   // UNICODE_TO_GBK[37326] := 16#941A;
   // UNICODE_TO_GBK[37327] := 16#E78C;
   // UNICODE_TO_GBK[37328] := 16#941B;
   // UNICODE_TO_GBK[37329] := 16#E78D;
   // UNICODE_TO_GBK[37330] := 16#941C;
   // UNICODE_TO_GBK[37331] := 16#E78E;
   // UNICODE_TO_GBK[37332] := 16#941D;
   // UNICODE_TO_GBK[37333] := 16#E78F;
   // UNICODE_TO_GBK[37334] := 16#941E;
   // UNICODE_TO_GBK[37335] := 16#E790;
   // UNICODE_TO_GBK[37336] := 16#941F;
   // UNICODE_TO_GBK[37337] := 16#E791;
   // UNICODE_TO_GBK[37338] := 16#9420;
   // UNICODE_TO_GBK[37339] := 16#E792;
   // UNICODE_TO_GBK[37340] := 16#9421;
   // UNICODE_TO_GBK[37341] := 16#E793;
   // UNICODE_TO_GBK[37342] := 16#9422;
   // UNICODE_TO_GBK[37343] := 16#E794;
   // UNICODE_TO_GBK[37344] := 16#9423;
   // UNICODE_TO_GBK[37345] := 16#E795;
   // UNICODE_TO_GBK[37346] := 16#9424;
   // UNICODE_TO_GBK[37347] := 16#E796;
   // UNICODE_TO_GBK[37348] := 16#9425;
   // UNICODE_TO_GBK[37349] := 16#E797;
   // UNICODE_TO_GBK[37350] := 16#9426;
   // UNICODE_TO_GBK[37351] := 16#E798;
   // UNICODE_TO_GBK[37352] := 16#9427;
   // UNICODE_TO_GBK[37353] := 16#E799;
   // UNICODE_TO_GBK[37354] := 16#9428;
   // UNICODE_TO_GBK[37355] := 16#E79A;
   // UNICODE_TO_GBK[37356] := 16#9429;
   // UNICODE_TO_GBK[37357] := 16#E79B;
   // UNICODE_TO_GBK[37358] := 16#942A;
   // UNICODE_TO_GBK[37359] := 16#E79C;
   // UNICODE_TO_GBK[37360] := 16#942B;
   // UNICODE_TO_GBK[37361] := 16#E79D;
   // UNICODE_TO_GBK[37362] := 16#942C;
   // UNICODE_TO_GBK[37363] := 16#E79E;
   // UNICODE_TO_GBK[37364] := 16#942D;
   // UNICODE_TO_GBK[37365] := 16#E79F;
   // UNICODE_TO_GBK[37366] := 16#942E;
   // UNICODE_TO_GBK[37367] := 16#E7A0;
   // UNICODE_TO_GBK[37368] := 16#942F;
   // UNICODE_TO_GBK[37369] := 16#E840;
   // UNICODE_TO_GBK[37370] := 16#9430;
   // UNICODE_TO_GBK[37371] := 16#E841;
   // UNICODE_TO_GBK[37372] := 16#9431;
   // UNICODE_TO_GBK[37373] := 16#E842;
   // UNICODE_TO_GBK[37374] := 16#9432;
   // UNICODE_TO_GBK[37375] := 16#E843;
   // UNICODE_TO_GBK[37376] := 16#9433;
   // UNICODE_TO_GBK[37377] := 16#E844;
   // UNICODE_TO_GBK[37378] := 16#9434;
   // UNICODE_TO_GBK[37379] := 16#E845;
   // UNICODE_TO_GBK[37380] := 16#9435;
   // UNICODE_TO_GBK[37381] := 16#E846;
   // UNICODE_TO_GBK[37382] := 16#9436;
   // UNICODE_TO_GBK[37383] := 16#E847;
   // UNICODE_TO_GBK[37384] := 16#9437;
   // UNICODE_TO_GBK[37385] := 16#E848;
   // UNICODE_TO_GBK[37386] := 16#9438;
   // UNICODE_TO_GBK[37387] := 16#E849;
   // UNICODE_TO_GBK[37388] := 16#9439;
   // UNICODE_TO_GBK[37389] := 16#E84A;
   // UNICODE_TO_GBK[37390] := 16#943A;
   // UNICODE_TO_GBK[37391] := 16#E84B;
   // UNICODE_TO_GBK[37392] := 16#943B;
   // UNICODE_TO_GBK[37393] := 16#E84C;
   // UNICODE_TO_GBK[37394] := 16#943C;
   // UNICODE_TO_GBK[37395] := 16#E84D;
   // UNICODE_TO_GBK[37396] := 16#943D;
   // UNICODE_TO_GBK[37397] := 16#E84E;
   // UNICODE_TO_GBK[37398] := 16#943E;
   // UNICODE_TO_GBK[37399] := 16#F6CD;
   // UNICODE_TO_GBK[37400] := 16#943F;
   // UNICODE_TO_GBK[37401] := 16#E84F;
   // UNICODE_TO_GBK[37402] := 16#9440;
   // UNICODE_TO_GBK[37403] := 16#E850;
   // UNICODE_TO_GBK[37404] := 16#9441;
   // UNICODE_TO_GBK[37405] := 16#E851;
   // UNICODE_TO_GBK[37406] := 16#9442;
   // UNICODE_TO_GBK[37407] := 16#E852;
   // UNICODE_TO_GBK[37408] := 16#9443;
   // UNICODE_TO_GBK[37409] := 16#E853;
   // UNICODE_TO_GBK[37410] := 16#9444;
   // UNICODE_TO_GBK[37411] := 16#E854;
   // UNICODE_TO_GBK[37412] := 16#9445;
   // UNICODE_TO_GBK[37413] := 16#E855;
   // UNICODE_TO_GBK[37414] := 16#9446;
   // UNICODE_TO_GBK[37415] := 16#E856;
   // UNICODE_TO_GBK[37416] := 16#9447;
   // UNICODE_TO_GBK[37417] := 16#E857;
   // UNICODE_TO_GBK[37418] := 16#9448;
   // UNICODE_TO_GBK[37419] := 16#E858;
   // UNICODE_TO_GBK[37420] := 16#9449;
   // UNICODE_TO_GBK[37421] := 16#E859;
   // UNICODE_TO_GBK[37422] := 16#944A;
   // UNICODE_TO_GBK[37423] := 16#E85A;
   // UNICODE_TO_GBK[37424] := 16#944B;
   // UNICODE_TO_GBK[37425] := 16#E85B;
   // UNICODE_TO_GBK[37426] := 16#944C;
   // UNICODE_TO_GBK[37427] := 16#E85C;
   // UNICODE_TO_GBK[37428] := 16#944D;
   // UNICODE_TO_GBK[37429] := 16#E85D;
   // UNICODE_TO_GBK[37430] := 16#944E;
   // UNICODE_TO_GBK[37431] := 16#E85E;
   // UNICODE_TO_GBK[37432] := 16#944F;
   // UNICODE_TO_GBK[37433] := 16#E85F;
   // UNICODE_TO_GBK[37434] := 16#9450;
   // UNICODE_TO_GBK[37435] := 16#E860;
   // UNICODE_TO_GBK[37436] := 16#9451;
   // UNICODE_TO_GBK[37437] := 16#E861;
   // UNICODE_TO_GBK[37438] := 16#9452;
   // UNICODE_TO_GBK[37439] := 16#E862;
   // UNICODE_TO_GBK[37440] := 16#9453;
   // UNICODE_TO_GBK[37441] := 16#E863;
   // UNICODE_TO_GBK[37442] := 16#9454;
   // UNICODE_TO_GBK[37443] := 16#E864;
   // UNICODE_TO_GBK[37444] := 16#9455;
   // UNICODE_TO_GBK[37445] := 16#E865;
   // UNICODE_TO_GBK[37446] := 16#9456;
   // UNICODE_TO_GBK[37447] := 16#E866;
   // UNICODE_TO_GBK[37448] := 16#9457;
   // UNICODE_TO_GBK[37449] := 16#E867;
   // UNICODE_TO_GBK[37450] := 16#9458;
   // UNICODE_TO_GBK[37451] := 16#E868;
   // UNICODE_TO_GBK[37452] := 16#9459;
   // UNICODE_TO_GBK[37453] := 16#E869;
   // UNICODE_TO_GBK[37454] := 16#945A;
   // UNICODE_TO_GBK[37455] := 16#E86A;
   // UNICODE_TO_GBK[37456] := 16#945B;
   // UNICODE_TO_GBK[37457] := 16#E86B;
   // UNICODE_TO_GBK[37458] := 16#945C;
   // UNICODE_TO_GBK[37459] := 16#E86C;
   // UNICODE_TO_GBK[37460] := 16#945D;
   // UNICODE_TO_GBK[37461] := 16#E86D;
   // UNICODE_TO_GBK[37462] := 16#945E;
   // UNICODE_TO_GBK[37463] := 16#E86E;
   // UNICODE_TO_GBK[37464] := 16#945F;
   // UNICODE_TO_GBK[37465] := 16#E86F;
   // UNICODE_TO_GBK[37466] := 16#9460;
   // UNICODE_TO_GBK[37467] := 16#E870;
   // UNICODE_TO_GBK[37468] := 16#9461;
   // UNICODE_TO_GBK[37469] := 16#E871;
   // UNICODE_TO_GBK[37470] := 16#9462;
   // UNICODE_TO_GBK[37471] := 16#E872;
   // UNICODE_TO_GBK[37472] := 16#9463;
   // UNICODE_TO_GBK[37473] := 16#E873;
   // UNICODE_TO_GBK[37474] := 16#9464;
   // UNICODE_TO_GBK[37475] := 16#E874;
   // UNICODE_TO_GBK[37476] := 16#9465;
   // UNICODE_TO_GBK[37477] := 16#E875;
   // UNICODE_TO_GBK[37478] := 16#9466;
   // UNICODE_TO_GBK[37479] := 16#E876;
   // UNICODE_TO_GBK[37480] := 16#9467;
   // UNICODE_TO_GBK[37481] := 16#E877;
   // UNICODE_TO_GBK[37482] := 16#9468;
   // UNICODE_TO_GBK[37483] := 16#E878;
   // UNICODE_TO_GBK[37484] := 16#9469;
   // UNICODE_TO_GBK[37485] := 16#E879;
   // UNICODE_TO_GBK[37486] := 16#946A;
   // UNICODE_TO_GBK[37487] := 16#E87A;
   // UNICODE_TO_GBK[37488] := 16#946B;
   // UNICODE_TO_GBK[37489] := 16#F6CE;
   // UNICODE_TO_GBK[37490] := 16#946C;
   // UNICODE_TO_GBK[37491] := 16#E87B;
   // UNICODE_TO_GBK[37492] := 16#946D;
   // UNICODE_TO_GBK[37493] := 16#E87C;
   // UNICODE_TO_GBK[37494] := 16#946E;
   // UNICODE_TO_GBK[37495] := 16#E87D;
   // UNICODE_TO_GBK[37496] := 16#946F;
   // UNICODE_TO_GBK[37497] := 16#E87E;
   // UNICODE_TO_GBK[37498] := 16#9470;
   // UNICODE_TO_GBK[37499] := 16#E880;
   // UNICODE_TO_GBK[37500] := 16#9471;
   // UNICODE_TO_GBK[37501] := 16#E881;
   // UNICODE_TO_GBK[37502] := 16#9472;
   // UNICODE_TO_GBK[37503] := 16#E882;
   // UNICODE_TO_GBK[37504] := 16#9473;
   // UNICODE_TO_GBK[37505] := 16#E883;
   // UNICODE_TO_GBK[37506] := 16#9474;
   // UNICODE_TO_GBK[37507] := 16#E884;
   // UNICODE_TO_GBK[37508] := 16#9475;
   // UNICODE_TO_GBK[37509] := 16#E885;
   // UNICODE_TO_GBK[37510] := 16#9476;
   // UNICODE_TO_GBK[37511] := 16#E886;
   // UNICODE_TO_GBK[37512] := 16#9477;
   // UNICODE_TO_GBK[37513] := 16#E887;
   // UNICODE_TO_GBK[37514] := 16#9478;
   // UNICODE_TO_GBK[37515] := 16#E888;
   // UNICODE_TO_GBK[37516] := 16#9479;
   // UNICODE_TO_GBK[37517] := 16#E889;
   // UNICODE_TO_GBK[37518] := 16#947A;
   // UNICODE_TO_GBK[37519] := 16#E88A;
   // UNICODE_TO_GBK[37520] := 16#947B;
   // UNICODE_TO_GBK[37521] := 16#E88B;
   // UNICODE_TO_GBK[37522] := 16#947C;
   // UNICODE_TO_GBK[37523] := 16#E88C;
   // UNICODE_TO_GBK[37524] := 16#947D;
   // UNICODE_TO_GBK[37525] := 16#E88D;
   // UNICODE_TO_GBK[37526] := 16#947E;
   // UNICODE_TO_GBK[37527] := 16#E88E;
   // UNICODE_TO_GBK[37528] := 16#947F;
   // UNICODE_TO_GBK[37529] := 16#E88F;
   // UNICODE_TO_GBK[37530] := 16#9480;
   // UNICODE_TO_GBK[37531] := 16#E890;
   // UNICODE_TO_GBK[37532] := 16#9481;
   // UNICODE_TO_GBK[37533] := 16#E891;
   // UNICODE_TO_GBK[37534] := 16#9482;
   // UNICODE_TO_GBK[37535] := 16#E892;
   // UNICODE_TO_GBK[37536] := 16#9483;
   // UNICODE_TO_GBK[37537] := 16#E893;
   // UNICODE_TO_GBK[37538] := 16#9484;
   // UNICODE_TO_GBK[37539] := 16#E894;
   // UNICODE_TO_GBK[37540] := 16#9485;
   // UNICODE_TO_GBK[37541] := 16#EEC4;
   // UNICODE_TO_GBK[37542] := 16#9486;
   // UNICODE_TO_GBK[37543] := 16#EEC5;
   // UNICODE_TO_GBK[37544] := 16#9487;
   // UNICODE_TO_GBK[37545] := 16#EEC6;
   // UNICODE_TO_GBK[37546] := 16#9488;
   // UNICODE_TO_GBK[37547] := 16#D5EB;
   // UNICODE_TO_GBK[37548] := 16#9489;
   // UNICODE_TO_GBK[37549] := 16#B6A4;
   // UNICODE_TO_GBK[37550] := 16#948A;
   // UNICODE_TO_GBK[37551] := 16#EEC8;
   // UNICODE_TO_GBK[37552] := 16#948B;
   // UNICODE_TO_GBK[37553] := 16#EEC7;
   // UNICODE_TO_GBK[37554] := 16#948C;
   // UNICODE_TO_GBK[37555] := 16#EEC9;
   // UNICODE_TO_GBK[37556] := 16#948D;
   // UNICODE_TO_GBK[37557] := 16#EECA;
   // UNICODE_TO_GBK[37558] := 16#948E;
   // UNICODE_TO_GBK[37559] := 16#C7A5;
   // UNICODE_TO_GBK[37560] := 16#948F;
   // UNICODE_TO_GBK[37561] := 16#EECB;
   // UNICODE_TO_GBK[37562] := 16#9490;
   // UNICODE_TO_GBK[37563] := 16#EECC;
   // UNICODE_TO_GBK[37564] := 16#9491;
   // UNICODE_TO_GBK[37565] := 16#E895;
   // UNICODE_TO_GBK[37566] := 16#9492;
   // UNICODE_TO_GBK[37567] := 16#B7B0;
   // UNICODE_TO_GBK[37568] := 16#9493;
   // UNICODE_TO_GBK[37569] := 16#B5F6;
   // UNICODE_TO_GBK[37570] := 16#9494;
   // UNICODE_TO_GBK[37571] := 16#EECD;
   // UNICODE_TO_GBK[37572] := 16#9495;
   // UNICODE_TO_GBK[37573] := 16#EECF;
   // UNICODE_TO_GBK[37574] := 16#9496;
   // UNICODE_TO_GBK[37575] := 16#E896;
   // UNICODE_TO_GBK[37576] := 16#9497;
   // UNICODE_TO_GBK[37577] := 16#EECE;
   // UNICODE_TO_GBK[37578] := 16#9498;
   // UNICODE_TO_GBK[37579] := 16#E897;
   // UNICODE_TO_GBK[37580] := 16#9499;
   // UNICODE_TO_GBK[37581] := 16#B8C6;
   // UNICODE_TO_GBK[37582] := 16#949A;
   // UNICODE_TO_GBK[37583] := 16#EED0;
   // UNICODE_TO_GBK[37584] := 16#949B;
   // UNICODE_TO_GBK[37585] := 16#EED1;
   // UNICODE_TO_GBK[37586] := 16#949C;
   // UNICODE_TO_GBK[37587] := 16#EED2;
   // UNICODE_TO_GBK[37588] := 16#949D;
   // UNICODE_TO_GBK[37589] := 16#B6DB;
   // UNICODE_TO_GBK[37590] := 16#949E;
   // UNICODE_TO_GBK[37591] := 16#B3AE;
   // UNICODE_TO_GBK[37592] := 16#949F;
   // UNICODE_TO_GBK[37593] := 16#D6D3;
   // UNICODE_TO_GBK[37594] := 16#94A0;
   // UNICODE_TO_GBK[37595] := 16#C4C6;
   // UNICODE_TO_GBK[37596] := 16#94A1;
   // UNICODE_TO_GBK[37597] := 16#B1B5;
   // UNICODE_TO_GBK[37598] := 16#94A2;
   // UNICODE_TO_GBK[37599] := 16#B8D6;
   // UNICODE_TO_GBK[37600] := 16#94A3;
   // UNICODE_TO_GBK[37601] := 16#EED3;
   // UNICODE_TO_GBK[37602] := 16#94A4;
   // UNICODE_TO_GBK[37603] := 16#EED4;
   // UNICODE_TO_GBK[37604] := 16#94A5;
   // UNICODE_TO_GBK[37605] := 16#D4BF;
   // UNICODE_TO_GBK[37606] := 16#94A6;
   // UNICODE_TO_GBK[37607] := 16#C7D5;
   // UNICODE_TO_GBK[37608] := 16#94A7;
   // UNICODE_TO_GBK[37609] := 16#BEFB;
   // UNICODE_TO_GBK[37610] := 16#94A8;
   // UNICODE_TO_GBK[37611] := 16#CED9;
   // UNICODE_TO_GBK[37612] := 16#94A9;
   // UNICODE_TO_GBK[37613] := 16#B9B3;
   // UNICODE_TO_GBK[37614] := 16#94AA;
   // UNICODE_TO_GBK[37615] := 16#EED6;
   // UNICODE_TO_GBK[37616] := 16#94AB;
   // UNICODE_TO_GBK[37617] := 16#EED5;
   // UNICODE_TO_GBK[37618] := 16#94AC;
   // UNICODE_TO_GBK[37619] := 16#EED8;
   // UNICODE_TO_GBK[37620] := 16#94AD;
   // UNICODE_TO_GBK[37621] := 16#EED7;
   // UNICODE_TO_GBK[37622] := 16#94AE;
   // UNICODE_TO_GBK[37623] := 16#C5A5;
   // UNICODE_TO_GBK[37624] := 16#94AF;
   // UNICODE_TO_GBK[37625] := 16#EED9;
   // UNICODE_TO_GBK[37626] := 16#94B0;
   // UNICODE_TO_GBK[37627] := 16#EEDA;
   // UNICODE_TO_GBK[37628] := 16#94B1;
   // UNICODE_TO_GBK[37629] := 16#C7AE;
   // UNICODE_TO_GBK[37630] := 16#94B2;
   // UNICODE_TO_GBK[37631] := 16#EEDB;
   // UNICODE_TO_GBK[37632] := 16#94B3;
   // UNICODE_TO_GBK[37633] := 16#C7AF;
   // UNICODE_TO_GBK[37634] := 16#94B4;
   // UNICODE_TO_GBK[37635] := 16#EEDC;
   // UNICODE_TO_GBK[37636] := 16#94B5;
   // UNICODE_TO_GBK[37637] := 16#B2A7;
   // UNICODE_TO_GBK[37638] := 16#94B6;
   // UNICODE_TO_GBK[37639] := 16#EEDD;
   // UNICODE_TO_GBK[37640] := 16#94B7;
   // UNICODE_TO_GBK[37641] := 16#EEDE;
   // UNICODE_TO_GBK[37642] := 16#94B8;
   // UNICODE_TO_GBK[37643] := 16#EEDF;
   // UNICODE_TO_GBK[37644] := 16#94B9;
   // UNICODE_TO_GBK[37645] := 16#EEE0;
   // UNICODE_TO_GBK[37646] := 16#94BA;
   // UNICODE_TO_GBK[37647] := 16#EEE1;
   // UNICODE_TO_GBK[37648] := 16#94BB;
   // UNICODE_TO_GBK[37649] := 16#D7EA;
   // UNICODE_TO_GBK[37650] := 16#94BC;
   // UNICODE_TO_GBK[37651] := 16#EEE2;
   // UNICODE_TO_GBK[37652] := 16#94BD;
   // UNICODE_TO_GBK[37653] := 16#EEE3;
   // UNICODE_TO_GBK[37654] := 16#94BE;
   // UNICODE_TO_GBK[37655] := 16#BCD8;
   // UNICODE_TO_GBK[37656] := 16#94BF;
   // UNICODE_TO_GBK[37657] := 16#EEE4;
   // UNICODE_TO_GBK[37658] := 16#94C0;
   // UNICODE_TO_GBK[37659] := 16#D3CB;
   // UNICODE_TO_GBK[37660] := 16#94C1;
   // UNICODE_TO_GBK[37661] := 16#CCFA;
   // UNICODE_TO_GBK[37662] := 16#94C2;
   // UNICODE_TO_GBK[37663] := 16#B2AC;
   // UNICODE_TO_GBK[37664] := 16#94C3;
   // UNICODE_TO_GBK[37665] := 16#C1E5;
   // UNICODE_TO_GBK[37666] := 16#94C4;
   // UNICODE_TO_GBK[37667] := 16#EEE5;
   // UNICODE_TO_GBK[37668] := 16#94C5;
   // UNICODE_TO_GBK[37669] := 16#C7A6;
   // UNICODE_TO_GBK[37670] := 16#94C6;
   // UNICODE_TO_GBK[37671] := 16#C3AD;
   // UNICODE_TO_GBK[37672] := 16#94C7;
   // UNICODE_TO_GBK[37673] := 16#E898;
   // UNICODE_TO_GBK[37674] := 16#94C8;
   // UNICODE_TO_GBK[37675] := 16#EEE6;
   // UNICODE_TO_GBK[37676] := 16#94C9;
   // UNICODE_TO_GBK[37677] := 16#EEE7;
   // UNICODE_TO_GBK[37678] := 16#94CA;
   // UNICODE_TO_GBK[37679] := 16#EEE8;
   // UNICODE_TO_GBK[37680] := 16#94CB;
   // UNICODE_TO_GBK[37681] := 16#EEE9;
   // UNICODE_TO_GBK[37682] := 16#94CC;
   // UNICODE_TO_GBK[37683] := 16#EEEA;
   // UNICODE_TO_GBK[37684] := 16#94CD;
   // UNICODE_TO_GBK[37685] := 16#EEEB;
   // UNICODE_TO_GBK[37686] := 16#94CE;
   // UNICODE_TO_GBK[37687] := 16#EEEC;
   // UNICODE_TO_GBK[37688] := 16#94CF;
   // UNICODE_TO_GBK[37689] := 16#E899;
   // UNICODE_TO_GBK[37690] := 16#94D0;
   // UNICODE_TO_GBK[37691] := 16#EEED;
   // UNICODE_TO_GBK[37692] := 16#94D1;
   // UNICODE_TO_GBK[37693] := 16#EEEE;
   // UNICODE_TO_GBK[37694] := 16#94D2;
   // UNICODE_TO_GBK[37695] := 16#EEEF;
   // UNICODE_TO_GBK[37696] := 16#94D3;
   // UNICODE_TO_GBK[37697] := 16#E89A;
   // UNICODE_TO_GBK[37698] := 16#94D4;
   // UNICODE_TO_GBK[37699] := 16#E89B;
   // UNICODE_TO_GBK[37700] := 16#94D5;
   // UNICODE_TO_GBK[37701] := 16#EEF0;
   // UNICODE_TO_GBK[37702] := 16#94D6;
   // UNICODE_TO_GBK[37703] := 16#EEF1;
   // UNICODE_TO_GBK[37704] := 16#94D7;
   // UNICODE_TO_GBK[37705] := 16#EEF2;
   // UNICODE_TO_GBK[37706] := 16#94D8;
   // UNICODE_TO_GBK[37707] := 16#EEF4;
   // UNICODE_TO_GBK[37708] := 16#94D9;
   // UNICODE_TO_GBK[37709] := 16#EEF3;
   // UNICODE_TO_GBK[37710] := 16#94DA;
   // UNICODE_TO_GBK[37711] := 16#E89C;
   // UNICODE_TO_GBK[37712] := 16#94DB;
   // UNICODE_TO_GBK[37713] := 16#EEF5;
   // UNICODE_TO_GBK[37714] := 16#94DC;
   // UNICODE_TO_GBK[37715] := 16#CDAD;
   // UNICODE_TO_GBK[37716] := 16#94DD;
   // UNICODE_TO_GBK[37717] := 16#C2C1;
   // UNICODE_TO_GBK[37718] := 16#94DE;
   // UNICODE_TO_GBK[37719] := 16#EEF6;
   // UNICODE_TO_GBK[37720] := 16#94DF;
   // UNICODE_TO_GBK[37721] := 16#EEF7;
   // UNICODE_TO_GBK[37722] := 16#94E0;
   // UNICODE_TO_GBK[37723] := 16#EEF8;
   // UNICODE_TO_GBK[37724] := 16#94E1;
   // UNICODE_TO_GBK[37725] := 16#D5A1;
   // UNICODE_TO_GBK[37726] := 16#94E2;
   // UNICODE_TO_GBK[37727] := 16#EEF9;
   // UNICODE_TO_GBK[37728] := 16#94E3;
   // UNICODE_TO_GBK[37729] := 16#CFB3;
   // UNICODE_TO_GBK[37730] := 16#94E4;
   // UNICODE_TO_GBK[37731] := 16#EEFA;
   // UNICODE_TO_GBK[37732] := 16#94E5;
   // UNICODE_TO_GBK[37733] := 16#EEFB;
   // UNICODE_TO_GBK[37734] := 16#94E6;
   // UNICODE_TO_GBK[37735] := 16#E89D;
   // UNICODE_TO_GBK[37736] := 16#94E7;
   // UNICODE_TO_GBK[37737] := 16#EEFC;
   // UNICODE_TO_GBK[37738] := 16#94E8;
   // UNICODE_TO_GBK[37739] := 16#EEFD;
   // UNICODE_TO_GBK[37740] := 16#94E9;
   // UNICODE_TO_GBK[37741] := 16#EFA1;
   // UNICODE_TO_GBK[37742] := 16#94EA;
   // UNICODE_TO_GBK[37743] := 16#EEFE;
   // UNICODE_TO_GBK[37744] := 16#94EB;
   // UNICODE_TO_GBK[37745] := 16#EFA2;
   // UNICODE_TO_GBK[37746] := 16#94EC;
   // UNICODE_TO_GBK[37747] := 16#B8F5;
   // UNICODE_TO_GBK[37748] := 16#94ED;
   // UNICODE_TO_GBK[37749] := 16#C3FA;
   // UNICODE_TO_GBK[37750] := 16#94EE;
   // UNICODE_TO_GBK[37751] := 16#EFA3;
   // UNICODE_TO_GBK[37752] := 16#94EF;
   // UNICODE_TO_GBK[37753] := 16#EFA4;
   // UNICODE_TO_GBK[37754] := 16#94F0;
   // UNICODE_TO_GBK[37755] := 16#BDC2;
   // UNICODE_TO_GBK[37756] := 16#94F1;
   // UNICODE_TO_GBK[37757] := 16#D2BF;
   // UNICODE_TO_GBK[37758] := 16#94F2;
   // UNICODE_TO_GBK[37759] := 16#B2F9;
   // UNICODE_TO_GBK[37760] := 16#94F3;
   // UNICODE_TO_GBK[37761] := 16#EFA5;
   // UNICODE_TO_GBK[37762] := 16#94F4;
   // UNICODE_TO_GBK[37763] := 16#EFA6;
   // UNICODE_TO_GBK[37764] := 16#94F5;
   // UNICODE_TO_GBK[37765] := 16#EFA7;
   // UNICODE_TO_GBK[37766] := 16#94F6;
   // UNICODE_TO_GBK[37767] := 16#D2F8;
   // UNICODE_TO_GBK[37768] := 16#94F7;
   // UNICODE_TO_GBK[37769] := 16#EFA8;
   // UNICODE_TO_GBK[37770] := 16#94F8;
   // UNICODE_TO_GBK[37771] := 16#D6FD;
   // UNICODE_TO_GBK[37772] := 16#94F9;
   // UNICODE_TO_GBK[37773] := 16#EFA9;
   // UNICODE_TO_GBK[37774] := 16#94FA;
   // UNICODE_TO_GBK[37775] := 16#C6CC;
   // UNICODE_TO_GBK[37776] := 16#94FB;
   // UNICODE_TO_GBK[37777] := 16#E89E;
   // UNICODE_TO_GBK[37778] := 16#94FC;
   // UNICODE_TO_GBK[37779] := 16#EFAA;
   // UNICODE_TO_GBK[37780] := 16#94FD;
   // UNICODE_TO_GBK[37781] := 16#EFAB;
   // UNICODE_TO_GBK[37782] := 16#94FE;
   // UNICODE_TO_GBK[37783] := 16#C1B4;
   // UNICODE_TO_GBK[37784] := 16#94FF;
   // UNICODE_TO_GBK[37785] := 16#EFAC;
   // UNICODE_TO_GBK[37786] := 16#9500;
   // UNICODE_TO_GBK[37787] := 16#CFFA;
   // UNICODE_TO_GBK[37788] := 16#9501;
   // UNICODE_TO_GBK[37789] := 16#CBF8;
   // UNICODE_TO_GBK[37790] := 16#9502;
   // UNICODE_TO_GBK[37791] := 16#EFAE;
   // UNICODE_TO_GBK[37792] := 16#9503;
   // UNICODE_TO_GBK[37793] := 16#EFAD;
   // UNICODE_TO_GBK[37794] := 16#9504;
   // UNICODE_TO_GBK[37795] := 16#B3FA;
   // UNICODE_TO_GBK[37796] := 16#9505;
   // UNICODE_TO_GBK[37797] := 16#B9F8;
   // UNICODE_TO_GBK[37798] := 16#9506;
   // UNICODE_TO_GBK[37799] := 16#EFAF;
   // UNICODE_TO_GBK[37800] := 16#9507;
   // UNICODE_TO_GBK[37801] := 16#EFB0;
   // UNICODE_TO_GBK[37802] := 16#9508;
   // UNICODE_TO_GBK[37803] := 16#D0E2;
   // UNICODE_TO_GBK[37804] := 16#9509;
   // UNICODE_TO_GBK[37805] := 16#EFB1;
   // UNICODE_TO_GBK[37806] := 16#950A;
   // UNICODE_TO_GBK[37807] := 16#EFB2;
   // UNICODE_TO_GBK[37808] := 16#950B;
   // UNICODE_TO_GBK[37809] := 16#B7E6;
   // UNICODE_TO_GBK[37810] := 16#950C;
   // UNICODE_TO_GBK[37811] := 16#D0BF;
   // UNICODE_TO_GBK[37812] := 16#950D;
   // UNICODE_TO_GBK[37813] := 16#EFB3;
   // UNICODE_TO_GBK[37814] := 16#950E;
   // UNICODE_TO_GBK[37815] := 16#EFB4;
   // UNICODE_TO_GBK[37816] := 16#950F;
   // UNICODE_TO_GBK[37817] := 16#EFB5;
   // UNICODE_TO_GBK[37818] := 16#9510;
   // UNICODE_TO_GBK[37819] := 16#C8F1;
   // UNICODE_TO_GBK[37820] := 16#9511;
   // UNICODE_TO_GBK[37821] := 16#CCE0;
   // UNICODE_TO_GBK[37822] := 16#9512;
   // UNICODE_TO_GBK[37823] := 16#EFB6;
   // UNICODE_TO_GBK[37824] := 16#9513;
   // UNICODE_TO_GBK[37825] := 16#EFB7;
   // UNICODE_TO_GBK[37826] := 16#9514;
   // UNICODE_TO_GBK[37827] := 16#EFB8;
   // UNICODE_TO_GBK[37828] := 16#9515;
   // UNICODE_TO_GBK[37829] := 16#EFB9;
   // UNICODE_TO_GBK[37830] := 16#9516;
   // UNICODE_TO_GBK[37831] := 16#EFBA;
   // UNICODE_TO_GBK[37832] := 16#9517;
   // UNICODE_TO_GBK[37833] := 16#D5E0;
   // UNICODE_TO_GBK[37834] := 16#9518;
   // UNICODE_TO_GBK[37835] := 16#EFBB;
   // UNICODE_TO_GBK[37836] := 16#9519;
   // UNICODE_TO_GBK[37837] := 16#B4ED;
   // UNICODE_TO_GBK[37838] := 16#951A;
   // UNICODE_TO_GBK[37839] := 16#C3AA;
   // UNICODE_TO_GBK[37840] := 16#951B;
   // UNICODE_TO_GBK[37841] := 16#EFBC;
   // UNICODE_TO_GBK[37842] := 16#951C;
   // UNICODE_TO_GBK[37843] := 16#E89F;
   // UNICODE_TO_GBK[37844] := 16#951D;
   // UNICODE_TO_GBK[37845] := 16#EFBD;
   // UNICODE_TO_GBK[37846] := 16#951E;
   // UNICODE_TO_GBK[37847] := 16#EFBE;
   // UNICODE_TO_GBK[37848] := 16#951F;
   // UNICODE_TO_GBK[37849] := 16#EFBF;
   // UNICODE_TO_GBK[37850] := 16#9520;
   // UNICODE_TO_GBK[37851] := 16#E8A0;
   // UNICODE_TO_GBK[37852] := 16#9521;
   // UNICODE_TO_GBK[37853] := 16#CEFD;
   // UNICODE_TO_GBK[37854] := 16#9522;
   // UNICODE_TO_GBK[37855] := 16#EFC0;
   // UNICODE_TO_GBK[37856] := 16#9523;
   // UNICODE_TO_GBK[37857] := 16#C2E0;
   // UNICODE_TO_GBK[37858] := 16#9524;
   // UNICODE_TO_GBK[37859] := 16#B4B8;
   // UNICODE_TO_GBK[37860] := 16#9525;
   // UNICODE_TO_GBK[37861] := 16#D7B6;
   // UNICODE_TO_GBK[37862] := 16#9526;
   // UNICODE_TO_GBK[37863] := 16#BDF5;
   // UNICODE_TO_GBK[37864] := 16#9527;
   // UNICODE_TO_GBK[37865] := 16#E940;
   // UNICODE_TO_GBK[37866] := 16#9528;
   // UNICODE_TO_GBK[37867] := 16#CFC7;
   // UNICODE_TO_GBK[37868] := 16#9529;
   // UNICODE_TO_GBK[37869] := 16#EFC3;
   // UNICODE_TO_GBK[37870] := 16#952A;
   // UNICODE_TO_GBK[37871] := 16#EFC1;
   // UNICODE_TO_GBK[37872] := 16#952B;
   // UNICODE_TO_GBK[37873] := 16#EFC2;
   // UNICODE_TO_GBK[37874] := 16#952C;
   // UNICODE_TO_GBK[37875] := 16#EFC4;
   // UNICODE_TO_GBK[37876] := 16#952D;
   // UNICODE_TO_GBK[37877] := 16#B6A7;
   // UNICODE_TO_GBK[37878] := 16#952E;
   // UNICODE_TO_GBK[37879] := 16#BCFC;
   // UNICODE_TO_GBK[37880] := 16#952F;
   // UNICODE_TO_GBK[37881] := 16#BEE2;
   // UNICODE_TO_GBK[37882] := 16#9530;
   // UNICODE_TO_GBK[37883] := 16#C3CC;
   // UNICODE_TO_GBK[37884] := 16#9531;
   // UNICODE_TO_GBK[37885] := 16#EFC5;
   // UNICODE_TO_GBK[37886] := 16#9532;
   // UNICODE_TO_GBK[37887] := 16#EFC6;
   // UNICODE_TO_GBK[37888] := 16#9533;
   // UNICODE_TO_GBK[37889] := 16#E941;
   // UNICODE_TO_GBK[37890] := 16#9534;
   // UNICODE_TO_GBK[37891] := 16#EFC7;
   // UNICODE_TO_GBK[37892] := 16#9535;
   // UNICODE_TO_GBK[37893] := 16#EFCF;
   // UNICODE_TO_GBK[37894] := 16#9536;
   // UNICODE_TO_GBK[37895] := 16#EFC8;
   // UNICODE_TO_GBK[37896] := 16#9537;
   // UNICODE_TO_GBK[37897] := 16#EFC9;
   // UNICODE_TO_GBK[37898] := 16#9538;
   // UNICODE_TO_GBK[37899] := 16#EFCA;
   // UNICODE_TO_GBK[37900] := 16#9539;
   // UNICODE_TO_GBK[37901] := 16#C7C2;
   // UNICODE_TO_GBK[37902] := 16#953A;
   // UNICODE_TO_GBK[37903] := 16#EFF1;
   // UNICODE_TO_GBK[37904] := 16#953B;
   // UNICODE_TO_GBK[37905] := 16#B6CD;
   // UNICODE_TO_GBK[37906] := 16#953C;
   // UNICODE_TO_GBK[37907] := 16#EFCB;
   // UNICODE_TO_GBK[37908] := 16#953D;
   // UNICODE_TO_GBK[37909] := 16#E942;
   // UNICODE_TO_GBK[37910] := 16#953E;
   // UNICODE_TO_GBK[37911] := 16#EFCC;
   // UNICODE_TO_GBK[37912] := 16#953F;
   // UNICODE_TO_GBK[37913] := 16#EFCD;
   // UNICODE_TO_GBK[37914] := 16#9540;
   // UNICODE_TO_GBK[37915] := 16#B6C6;
   // UNICODE_TO_GBK[37916] := 16#9541;
   // UNICODE_TO_GBK[37917] := 16#C3BE;
   // UNICODE_TO_GBK[37918] := 16#9542;
   // UNICODE_TO_GBK[37919] := 16#EFCE;
   // UNICODE_TO_GBK[37920] := 16#9543;
   // UNICODE_TO_GBK[37921] := 16#E943;
   // UNICODE_TO_GBK[37922] := 16#9544;
   // UNICODE_TO_GBK[37923] := 16#EFD0;
   // UNICODE_TO_GBK[37924] := 16#9545;
   // UNICODE_TO_GBK[37925] := 16#EFD1;
   // UNICODE_TO_GBK[37926] := 16#9546;
   // UNICODE_TO_GBK[37927] := 16#EFD2;
   // UNICODE_TO_GBK[37928] := 16#9547;
   // UNICODE_TO_GBK[37929] := 16#D5F2;
   // UNICODE_TO_GBK[37930] := 16#9548;
   // UNICODE_TO_GBK[37931] := 16#E944;
   // UNICODE_TO_GBK[37932] := 16#9549;
   // UNICODE_TO_GBK[37933] := 16#EFD3;
   // UNICODE_TO_GBK[37934] := 16#954A;
   // UNICODE_TO_GBK[37935] := 16#C4F7;
   // UNICODE_TO_GBK[37936] := 16#954B;
   // UNICODE_TO_GBK[37937] := 16#E945;
   // UNICODE_TO_GBK[37938] := 16#954C;
   // UNICODE_TO_GBK[37939] := 16#EFD4;
   // UNICODE_TO_GBK[37940] := 16#954D;
   // UNICODE_TO_GBK[37941] := 16#C4F8;
   // UNICODE_TO_GBK[37942] := 16#954E;
   // UNICODE_TO_GBK[37943] := 16#EFD5;
   // UNICODE_TO_GBK[37944] := 16#954F;
   // UNICODE_TO_GBK[37945] := 16#EFD6;
   // UNICODE_TO_GBK[37946] := 16#9550;
   // UNICODE_TO_GBK[37947] := 16#B8E4;
   // UNICODE_TO_GBK[37948] := 16#9551;
   // UNICODE_TO_GBK[37949] := 16#B0F7;
   // UNICODE_TO_GBK[37950] := 16#9552;
   // UNICODE_TO_GBK[37951] := 16#EFD7;
   // UNICODE_TO_GBK[37952] := 16#9553;
   // UNICODE_TO_GBK[37953] := 16#EFD8;
   // UNICODE_TO_GBK[37954] := 16#9554;
   // UNICODE_TO_GBK[37955] := 16#EFD9;
   // UNICODE_TO_GBK[37956] := 16#9555;
   // UNICODE_TO_GBK[37957] := 16#E946;
   // UNICODE_TO_GBK[37958] := 16#9556;
   // UNICODE_TO_GBK[37959] := 16#EFDA;
   // UNICODE_TO_GBK[37960] := 16#9557;
   // UNICODE_TO_GBK[37961] := 16#EFDB;
   // UNICODE_TO_GBK[37962] := 16#9558;
   // UNICODE_TO_GBK[37963] := 16#EFDC;
   // UNICODE_TO_GBK[37964] := 16#9559;
   // UNICODE_TO_GBK[37965] := 16#EFDD;
   // UNICODE_TO_GBK[37966] := 16#955A;
   // UNICODE_TO_GBK[37967] := 16#E947;
   // UNICODE_TO_GBK[37968] := 16#955B;
   // UNICODE_TO_GBK[37969] := 16#EFDE;
   // UNICODE_TO_GBK[37970] := 16#955C;
   // UNICODE_TO_GBK[37971] := 16#BEB5;
   // UNICODE_TO_GBK[37972] := 16#955D;
   // UNICODE_TO_GBK[37973] := 16#EFE1;
   // UNICODE_TO_GBK[37974] := 16#955E;
   // UNICODE_TO_GBK[37975] := 16#EFDF;
   // UNICODE_TO_GBK[37976] := 16#955F;
   // UNICODE_TO_GBK[37977] := 16#EFE0;
   // UNICODE_TO_GBK[37978] := 16#9560;
   // UNICODE_TO_GBK[37979] := 16#E948;
   // UNICODE_TO_GBK[37980] := 16#9561;
   // UNICODE_TO_GBK[37981] := 16#EFE2;
   // UNICODE_TO_GBK[37982] := 16#9562;
   // UNICODE_TO_GBK[37983] := 16#EFE3;
   // UNICODE_TO_GBK[37984] := 16#9563;
   // UNICODE_TO_GBK[37985] := 16#C1CD;
   // UNICODE_TO_GBK[37986] := 16#9564;
   // UNICODE_TO_GBK[37987] := 16#EFE4;
   // UNICODE_TO_GBK[37988] := 16#9565;
   // UNICODE_TO_GBK[37989] := 16#EFE5;
   // UNICODE_TO_GBK[37990] := 16#9566;
   // UNICODE_TO_GBK[37991] := 16#EFE6;
   // UNICODE_TO_GBK[37992] := 16#9567;
   // UNICODE_TO_GBK[37993] := 16#EFE7;
   // UNICODE_TO_GBK[37994] := 16#9568;
   // UNICODE_TO_GBK[37995] := 16#EFE8;
   // UNICODE_TO_GBK[37996] := 16#9569;
   // UNICODE_TO_GBK[37997] := 16#EFE9;
   // UNICODE_TO_GBK[37998] := 16#956A;
   // UNICODE_TO_GBK[37999] := 16#EFEA;
   // UNICODE_TO_GBK[38000] := 16#956B;
   // UNICODE_TO_GBK[38001] := 16#EFEB;
   // UNICODE_TO_GBK[38002] := 16#956C;
   // UNICODE_TO_GBK[38003] := 16#EFEC;
   // UNICODE_TO_GBK[38004] := 16#956D;
   // UNICODE_TO_GBK[38005] := 16#C0D8;
   // UNICODE_TO_GBK[38006] := 16#956E;
   // UNICODE_TO_GBK[38007] := 16#E949;
   // UNICODE_TO_GBK[38008] := 16#956F;
   // UNICODE_TO_GBK[38009] := 16#EFED;
   // UNICODE_TO_GBK[38010] := 16#9570;
   // UNICODE_TO_GBK[38011] := 16#C1AD;
   // UNICODE_TO_GBK[38012] := 16#9571;
   // UNICODE_TO_GBK[38013] := 16#EFEE;
   // UNICODE_TO_GBK[38014] := 16#9572;
   // UNICODE_TO_GBK[38015] := 16#EFEF;
   // UNICODE_TO_GBK[38016] := 16#9573;
   // UNICODE_TO_GBK[38017] := 16#EFF0;
   // UNICODE_TO_GBK[38018] := 16#9574;
   // UNICODE_TO_GBK[38019] := 16#E94A;
   // UNICODE_TO_GBK[38020] := 16#9575;
   // UNICODE_TO_GBK[38021] := 16#E94B;
   // UNICODE_TO_GBK[38022] := 16#9576;
   // UNICODE_TO_GBK[38023] := 16#CFE2;
   // UNICODE_TO_GBK[38024] := 16#9577;
   // UNICODE_TO_GBK[38025] := 16#E94C;
   // UNICODE_TO_GBK[38026] := 16#9578;
   // UNICODE_TO_GBK[38027] := 16#E94D;
   // UNICODE_TO_GBK[38028] := 16#9579;
   // UNICODE_TO_GBK[38029] := 16#E94E;
   // UNICODE_TO_GBK[38030] := 16#957A;
   // UNICODE_TO_GBK[38031] := 16#E94F;
   // UNICODE_TO_GBK[38032] := 16#957B;
   // UNICODE_TO_GBK[38033] := 16#E950;
   // UNICODE_TO_GBK[38034] := 16#957C;
   // UNICODE_TO_GBK[38035] := 16#E951;
   // UNICODE_TO_GBK[38036] := 16#957D;
   // UNICODE_TO_GBK[38037] := 16#E952;
   // UNICODE_TO_GBK[38038] := 16#957E;
   // UNICODE_TO_GBK[38039] := 16#E953;
   // UNICODE_TO_GBK[38040] := 16#957F;
   // UNICODE_TO_GBK[38041] := 16#B3A4;
   // UNICODE_TO_GBK[38042] := 16#9580;
   // UNICODE_TO_GBK[38043] := 16#E954;
   // UNICODE_TO_GBK[38044] := 16#9581;
   // UNICODE_TO_GBK[38045] := 16#E955;
   // UNICODE_TO_GBK[38046] := 16#9582;
   // UNICODE_TO_GBK[38047] := 16#E956;
   // UNICODE_TO_GBK[38048] := 16#9583;
   // UNICODE_TO_GBK[38049] := 16#E957;
   // UNICODE_TO_GBK[38050] := 16#9584;
   // UNICODE_TO_GBK[38051] := 16#E958;
   // UNICODE_TO_GBK[38052] := 16#9585;
   // UNICODE_TO_GBK[38053] := 16#E959;
   // UNICODE_TO_GBK[38054] := 16#9586;
   // UNICODE_TO_GBK[38055] := 16#E95A;
   // UNICODE_TO_GBK[38056] := 16#9587;
   // UNICODE_TO_GBK[38057] := 16#E95B;
   // UNICODE_TO_GBK[38058] := 16#9588;
   // UNICODE_TO_GBK[38059] := 16#E95C;
   // UNICODE_TO_GBK[38060] := 16#9589;
   // UNICODE_TO_GBK[38061] := 16#E95D;
   // UNICODE_TO_GBK[38062] := 16#958A;
   // UNICODE_TO_GBK[38063] := 16#E95E;
   // UNICODE_TO_GBK[38064] := 16#958B;
   // UNICODE_TO_GBK[38065] := 16#E95F;
   // UNICODE_TO_GBK[38066] := 16#958C;
   // UNICODE_TO_GBK[38067] := 16#E960;
   // UNICODE_TO_GBK[38068] := 16#958D;
   // UNICODE_TO_GBK[38069] := 16#E961;
   // UNICODE_TO_GBK[38070] := 16#958E;
   // UNICODE_TO_GBK[38071] := 16#E962;
   // UNICODE_TO_GBK[38072] := 16#958F;
   // UNICODE_TO_GBK[38073] := 16#E963;
   // UNICODE_TO_GBK[38074] := 16#9590;
   // UNICODE_TO_GBK[38075] := 16#E964;
   // UNICODE_TO_GBK[38076] := 16#9591;
   // UNICODE_TO_GBK[38077] := 16#E965;
   // UNICODE_TO_GBK[38078] := 16#9592;
   // UNICODE_TO_GBK[38079] := 16#E966;
   // UNICODE_TO_GBK[38080] := 16#9593;
   // UNICODE_TO_GBK[38081] := 16#E967;
   // UNICODE_TO_GBK[38082] := 16#9594;
   // UNICODE_TO_GBK[38083] := 16#E968;
   // UNICODE_TO_GBK[38084] := 16#9595;
   // UNICODE_TO_GBK[38085] := 16#E969;
   // UNICODE_TO_GBK[38086] := 16#9596;
   // UNICODE_TO_GBK[38087] := 16#E96A;
   // UNICODE_TO_GBK[38088] := 16#9597;
   // UNICODE_TO_GBK[38089] := 16#E96B;
   // UNICODE_TO_GBK[38090] := 16#9598;
   // UNICODE_TO_GBK[38091] := 16#E96C;
   // UNICODE_TO_GBK[38092] := 16#9599;
   // UNICODE_TO_GBK[38093] := 16#E96D;
   // UNICODE_TO_GBK[38094] := 16#959A;
   // UNICODE_TO_GBK[38095] := 16#E96E;
   // UNICODE_TO_GBK[38096] := 16#959B;
   // UNICODE_TO_GBK[38097] := 16#E96F;
   // UNICODE_TO_GBK[38098] := 16#959C;
   // UNICODE_TO_GBK[38099] := 16#E970;
   // UNICODE_TO_GBK[38100] := 16#959D;
   // UNICODE_TO_GBK[38101] := 16#E971;
   // UNICODE_TO_GBK[38102] := 16#959E;
   // UNICODE_TO_GBK[38103] := 16#E972;
   // UNICODE_TO_GBK[38104] := 16#959F;
   // UNICODE_TO_GBK[38105] := 16#E973;
   // UNICODE_TO_GBK[38106] := 16#95A0;
   // UNICODE_TO_GBK[38107] := 16#E974;
   // UNICODE_TO_GBK[38108] := 16#95A1;
   // UNICODE_TO_GBK[38109] := 16#E975;
   // UNICODE_TO_GBK[38110] := 16#95A2;
   // UNICODE_TO_GBK[38111] := 16#E976;
   // UNICODE_TO_GBK[38112] := 16#95A3;
   // UNICODE_TO_GBK[38113] := 16#E977;
   // UNICODE_TO_GBK[38114] := 16#95A4;
   // UNICODE_TO_GBK[38115] := 16#E978;
   // UNICODE_TO_GBK[38116] := 16#95A5;
   // UNICODE_TO_GBK[38117] := 16#E979;
   // UNICODE_TO_GBK[38118] := 16#95A6;
   // UNICODE_TO_GBK[38119] := 16#E97A;
   // UNICODE_TO_GBK[38120] := 16#95A7;
   // UNICODE_TO_GBK[38121] := 16#E97B;
   // UNICODE_TO_GBK[38122] := 16#95A8;
   // UNICODE_TO_GBK[38123] := 16#E97C;
   // UNICODE_TO_GBK[38124] := 16#95A9;
   // UNICODE_TO_GBK[38125] := 16#E97D;
   // UNICODE_TO_GBK[38126] := 16#95AA;
   // UNICODE_TO_GBK[38127] := 16#E97E;
   // UNICODE_TO_GBK[38128] := 16#95AB;
   // UNICODE_TO_GBK[38129] := 16#E980;
   // UNICODE_TO_GBK[38130] := 16#95AC;
   // UNICODE_TO_GBK[38131] := 16#E981;
   // UNICODE_TO_GBK[38132] := 16#95AD;
   // UNICODE_TO_GBK[38133] := 16#E982;
   // UNICODE_TO_GBK[38134] := 16#95AE;
   // UNICODE_TO_GBK[38135] := 16#E983;
   // UNICODE_TO_GBK[38136] := 16#95AF;
   // UNICODE_TO_GBK[38137] := 16#E984;
   // UNICODE_TO_GBK[38138] := 16#95B0;
   // UNICODE_TO_GBK[38139] := 16#E985;
   // UNICODE_TO_GBK[38140] := 16#95B1;
   // UNICODE_TO_GBK[38141] := 16#E986;
   // UNICODE_TO_GBK[38142] := 16#95B2;
   // UNICODE_TO_GBK[38143] := 16#E987;
   // UNICODE_TO_GBK[38144] := 16#95B3;
   // UNICODE_TO_GBK[38145] := 16#E988;
   // UNICODE_TO_GBK[38146] := 16#95B4;
   // UNICODE_TO_GBK[38147] := 16#E989;
   // UNICODE_TO_GBK[38148] := 16#95B5;
   // UNICODE_TO_GBK[38149] := 16#E98A;
   // UNICODE_TO_GBK[38150] := 16#95B6;
   // UNICODE_TO_GBK[38151] := 16#E98B;
   // UNICODE_TO_GBK[38152] := 16#95B7;
   // UNICODE_TO_GBK[38153] := 16#E98C;
   // UNICODE_TO_GBK[38154] := 16#95B8;
   // UNICODE_TO_GBK[38155] := 16#E98D;
   // UNICODE_TO_GBK[38156] := 16#95B9;
   // UNICODE_TO_GBK[38157] := 16#E98E;
   // UNICODE_TO_GBK[38158] := 16#95BA;
   // UNICODE_TO_GBK[38159] := 16#E98F;
   // UNICODE_TO_GBK[38160] := 16#95BB;
   // UNICODE_TO_GBK[38161] := 16#E990;
   // UNICODE_TO_GBK[38162] := 16#95BC;
   // UNICODE_TO_GBK[38163] := 16#E991;
   // UNICODE_TO_GBK[38164] := 16#95BD;
   // UNICODE_TO_GBK[38165] := 16#E992;
   // UNICODE_TO_GBK[38166] := 16#95BE;
   // UNICODE_TO_GBK[38167] := 16#E993;
   // UNICODE_TO_GBK[38168] := 16#95BF;
   // UNICODE_TO_GBK[38169] := 16#E994;
   // UNICODE_TO_GBK[38170] := 16#95C0;
   // UNICODE_TO_GBK[38171] := 16#E995;
   // UNICODE_TO_GBK[38172] := 16#95C1;
   // UNICODE_TO_GBK[38173] := 16#E996;
   // UNICODE_TO_GBK[38174] := 16#95C2;
   // UNICODE_TO_GBK[38175] := 16#E997;
   // UNICODE_TO_GBK[38176] := 16#95C3;
   // UNICODE_TO_GBK[38177] := 16#E998;
   // UNICODE_TO_GBK[38178] := 16#95C4;
   // UNICODE_TO_GBK[38179] := 16#E999;
   // UNICODE_TO_GBK[38180] := 16#95C5;
   // UNICODE_TO_GBK[38181] := 16#E99A;
   // UNICODE_TO_GBK[38182] := 16#95C6;
   // UNICODE_TO_GBK[38183] := 16#E99B;
   // UNICODE_TO_GBK[38184] := 16#95C7;
   // UNICODE_TO_GBK[38185] := 16#E99C;
   // UNICODE_TO_GBK[38186] := 16#95C8;
   // UNICODE_TO_GBK[38187] := 16#E99D;
   // UNICODE_TO_GBK[38188] := 16#95C9;
   // UNICODE_TO_GBK[38189] := 16#E99E;
   // UNICODE_TO_GBK[38190] := 16#95CA;
   // UNICODE_TO_GBK[38191] := 16#E99F;
   // UNICODE_TO_GBK[38192] := 16#95CB;
   // UNICODE_TO_GBK[38193] := 16#E9A0;
   // UNICODE_TO_GBK[38194] := 16#95CC;
   // UNICODE_TO_GBK[38195] := 16#EA40;
   // UNICODE_TO_GBK[38196] := 16#95CD;
   // UNICODE_TO_GBK[38197] := 16#EA41;
   // UNICODE_TO_GBK[38198] := 16#95CE;
   // UNICODE_TO_GBK[38199] := 16#EA42;
   // UNICODE_TO_GBK[38200] := 16#95CF;
   // UNICODE_TO_GBK[38201] := 16#EA43;
   // UNICODE_TO_GBK[38202] := 16#95D0;
   // UNICODE_TO_GBK[38203] := 16#EA44;
   // UNICODE_TO_GBK[38204] := 16#95D1;
   // UNICODE_TO_GBK[38205] := 16#EA45;
   // UNICODE_TO_GBK[38206] := 16#95D2;
   // UNICODE_TO_GBK[38207] := 16#EA46;
   // UNICODE_TO_GBK[38208] := 16#95D3;
   // UNICODE_TO_GBK[38209] := 16#EA47;
   // UNICODE_TO_GBK[38210] := 16#95D4;
   // UNICODE_TO_GBK[38211] := 16#EA48;
   // UNICODE_TO_GBK[38212] := 16#95D5;
   // UNICODE_TO_GBK[38213] := 16#EA49;
   // UNICODE_TO_GBK[38214] := 16#95D6;
   // UNICODE_TO_GBK[38215] := 16#EA4A;
   // UNICODE_TO_GBK[38216] := 16#95D7;
   // UNICODE_TO_GBK[38217] := 16#EA4B;
   // UNICODE_TO_GBK[38218] := 16#95D8;
   // UNICODE_TO_GBK[38219] := 16#EA4C;
   // UNICODE_TO_GBK[38220] := 16#95D9;
   // UNICODE_TO_GBK[38221] := 16#EA4D;
   // UNICODE_TO_GBK[38222] := 16#95DA;
   // UNICODE_TO_GBK[38223] := 16#EA4E;
   // UNICODE_TO_GBK[38224] := 16#95DB;
   // UNICODE_TO_GBK[38225] := 16#EA4F;
   // UNICODE_TO_GBK[38226] := 16#95DC;
   // UNICODE_TO_GBK[38227] := 16#EA50;
   // UNICODE_TO_GBK[38228] := 16#95DD;
   // UNICODE_TO_GBK[38229] := 16#EA51;
   // UNICODE_TO_GBK[38230] := 16#95DE;
   // UNICODE_TO_GBK[38231] := 16#EA52;
   // UNICODE_TO_GBK[38232] := 16#95DF;
   // UNICODE_TO_GBK[38233] := 16#EA53;
   // UNICODE_TO_GBK[38234] := 16#95E0;
   // UNICODE_TO_GBK[38235] := 16#EA54;
   // UNICODE_TO_GBK[38236] := 16#95E1;
   // UNICODE_TO_GBK[38237] := 16#EA55;
   // UNICODE_TO_GBK[38238] := 16#95E2;
   // UNICODE_TO_GBK[38239] := 16#EA56;
   // UNICODE_TO_GBK[38240] := 16#95E3;
   // UNICODE_TO_GBK[38241] := 16#EA57;
   // UNICODE_TO_GBK[38242] := 16#95E4;
   // UNICODE_TO_GBK[38243] := 16#EA58;
   // UNICODE_TO_GBK[38244] := 16#95E5;
   // UNICODE_TO_GBK[38245] := 16#EA59;
   // UNICODE_TO_GBK[38246] := 16#95E6;
   // UNICODE_TO_GBK[38247] := 16#EA5A;
   // UNICODE_TO_GBK[38248] := 16#95E7;
   // UNICODE_TO_GBK[38249] := 16#EA5B;
   // UNICODE_TO_GBK[38250] := 16#95E8;
   // UNICODE_TO_GBK[38251] := 16#C3C5;
   // UNICODE_TO_GBK[38252] := 16#95E9;
   // UNICODE_TO_GBK[38253] := 16#E3C5;
   // UNICODE_TO_GBK[38254] := 16#95EA;
   // UNICODE_TO_GBK[38255] := 16#C9C1;
   // UNICODE_TO_GBK[38256] := 16#95EB;
   // UNICODE_TO_GBK[38257] := 16#E3C6;
   // UNICODE_TO_GBK[38258] := 16#95EC;
   // UNICODE_TO_GBK[38259] := 16#EA5C;
   // UNICODE_TO_GBK[38260] := 16#95ED;
   // UNICODE_TO_GBK[38261] := 16#B1D5;
   // UNICODE_TO_GBK[38262] := 16#95EE;
   // UNICODE_TO_GBK[38263] := 16#CECA;
   // UNICODE_TO_GBK[38264] := 16#95EF;
   // UNICODE_TO_GBK[38265] := 16#B4B3;
   // UNICODE_TO_GBK[38266] := 16#95F0;
   // UNICODE_TO_GBK[38267] := 16#C8F2;
   // UNICODE_TO_GBK[38268] := 16#95F1;
   // UNICODE_TO_GBK[38269] := 16#E3C7;
   // UNICODE_TO_GBK[38270] := 16#95F2;
   // UNICODE_TO_GBK[38271] := 16#CFD0;
   // UNICODE_TO_GBK[38272] := 16#95F3;
   // UNICODE_TO_GBK[38273] := 16#E3C8;
   // UNICODE_TO_GBK[38274] := 16#95F4;
   // UNICODE_TO_GBK[38275] := 16#BCE4;
   // UNICODE_TO_GBK[38276] := 16#95F5;
   // UNICODE_TO_GBK[38277] := 16#E3C9;
   // UNICODE_TO_GBK[38278] := 16#95F6;
   // UNICODE_TO_GBK[38279] := 16#E3CA;
   // UNICODE_TO_GBK[38280] := 16#95F7;
   // UNICODE_TO_GBK[38281] := 16#C3C6;
   // UNICODE_TO_GBK[38282] := 16#95F8;
   // UNICODE_TO_GBK[38283] := 16#D5A2;
   // UNICODE_TO_GBK[38284] := 16#95F9;
   // UNICODE_TO_GBK[38285] := 16#C4D6;
   // UNICODE_TO_GBK[38286] := 16#95FA;
   // UNICODE_TO_GBK[38287] := 16#B9EB;
   // UNICODE_TO_GBK[38288] := 16#95FB;
   // UNICODE_TO_GBK[38289] := 16#CEC5;
   // UNICODE_TO_GBK[38290] := 16#95FC;
   // UNICODE_TO_GBK[38291] := 16#E3CB;
   // UNICODE_TO_GBK[38292] := 16#95FD;
   // UNICODE_TO_GBK[38293] := 16#C3F6;
   // UNICODE_TO_GBK[38294] := 16#95FE;
   // UNICODE_TO_GBK[38295] := 16#E3CC;
   // UNICODE_TO_GBK[38296] := 16#95FF;
   // UNICODE_TO_GBK[38297] := 16#EA5D;
   // UNICODE_TO_GBK[38298] := 16#9600;
   // UNICODE_TO_GBK[38299] := 16#B7A7;
   // UNICODE_TO_GBK[38300] := 16#9601;
   // UNICODE_TO_GBK[38301] := 16#B8F3;
   // UNICODE_TO_GBK[38302] := 16#9602;
   // UNICODE_TO_GBK[38303] := 16#BAD2;
   // UNICODE_TO_GBK[38304] := 16#9603;
   // UNICODE_TO_GBK[38305] := 16#E3CD;
   // UNICODE_TO_GBK[38306] := 16#9604;
   // UNICODE_TO_GBK[38307] := 16#E3CE;
   // UNICODE_TO_GBK[38308] := 16#9605;
   // UNICODE_TO_GBK[38309] := 16#D4C4;
   // UNICODE_TO_GBK[38310] := 16#9606;
   // UNICODE_TO_GBK[38311] := 16#E3CF;
   // UNICODE_TO_GBK[38312] := 16#9607;
   // UNICODE_TO_GBK[38313] := 16#EA5E;
   // UNICODE_TO_GBK[38314] := 16#9608;
   // UNICODE_TO_GBK[38315] := 16#E3D0;
   // UNICODE_TO_GBK[38316] := 16#9609;
   // UNICODE_TO_GBK[38317] := 16#D1CB;
   // UNICODE_TO_GBK[38318] := 16#960A;
   // UNICODE_TO_GBK[38319] := 16#E3D1;
   // UNICODE_TO_GBK[38320] := 16#960B;
   // UNICODE_TO_GBK[38321] := 16#E3D2;
   // UNICODE_TO_GBK[38322] := 16#960C;
   // UNICODE_TO_GBK[38323] := 16#E3D3;
   // UNICODE_TO_GBK[38324] := 16#960D;
   // UNICODE_TO_GBK[38325] := 16#E3D4;
   // UNICODE_TO_GBK[38326] := 16#960E;
   // UNICODE_TO_GBK[38327] := 16#D1D6;
   // UNICODE_TO_GBK[38328] := 16#960F;
   // UNICODE_TO_GBK[38329] := 16#E3D5;
   // UNICODE_TO_GBK[38330] := 16#9610;
   // UNICODE_TO_GBK[38331] := 16#B2FB;
   // UNICODE_TO_GBK[38332] := 16#9611;
   // UNICODE_TO_GBK[38333] := 16#C0BB;
   // UNICODE_TO_GBK[38334] := 16#9612;
   // UNICODE_TO_GBK[38335] := 16#E3D6;
   // UNICODE_TO_GBK[38336] := 16#9613;
   // UNICODE_TO_GBK[38337] := 16#EA5F;
   // UNICODE_TO_GBK[38338] := 16#9614;
   // UNICODE_TO_GBK[38339] := 16#C0AB;
   // UNICODE_TO_GBK[38340] := 16#9615;
   // UNICODE_TO_GBK[38341] := 16#E3D7;
   // UNICODE_TO_GBK[38342] := 16#9616;
   // UNICODE_TO_GBK[38343] := 16#E3D8;
   // UNICODE_TO_GBK[38344] := 16#9617;
   // UNICODE_TO_GBK[38345] := 16#E3D9;
   // UNICODE_TO_GBK[38346] := 16#9618;
   // UNICODE_TO_GBK[38347] := 16#EA60;
   // UNICODE_TO_GBK[38348] := 16#9619;
   // UNICODE_TO_GBK[38349] := 16#E3DA;
   // UNICODE_TO_GBK[38350] := 16#961A;
   // UNICODE_TO_GBK[38351] := 16#E3DB;
   // UNICODE_TO_GBK[38352] := 16#961B;
   // UNICODE_TO_GBK[38353] := 16#EA61;
   // UNICODE_TO_GBK[38354] := 16#961C;
   // UNICODE_TO_GBK[38355] := 16#B8B7;
   // UNICODE_TO_GBK[38356] := 16#961D;
   // UNICODE_TO_GBK[38357] := 16#DAE2;
   // UNICODE_TO_GBK[38358] := 16#961E;
   // UNICODE_TO_GBK[38359] := 16#EA62;
   // UNICODE_TO_GBK[38360] := 16#961F;
   // UNICODE_TO_GBK[38361] := 16#B6D3;
   // UNICODE_TO_GBK[38362] := 16#9620;
   // UNICODE_TO_GBK[38363] := 16#EA63;
   // UNICODE_TO_GBK[38364] := 16#9621;
   // UNICODE_TO_GBK[38365] := 16#DAE4;
   // UNICODE_TO_GBK[38366] := 16#9622;
   // UNICODE_TO_GBK[38367] := 16#DAE3;
   // UNICODE_TO_GBK[38368] := 16#9623;
   // UNICODE_TO_GBK[38369] := 16#EA64;
   // UNICODE_TO_GBK[38370] := 16#9624;
   // UNICODE_TO_GBK[38371] := 16#EA65;
   // UNICODE_TO_GBK[38372] := 16#9625;
   // UNICODE_TO_GBK[38373] := 16#EA66;
   // UNICODE_TO_GBK[38374] := 16#9626;
   // UNICODE_TO_GBK[38375] := 16#EA67;
   // UNICODE_TO_GBK[38376] := 16#9627;
   // UNICODE_TO_GBK[38377] := 16#EA68;
   // UNICODE_TO_GBK[38378] := 16#9628;
   // UNICODE_TO_GBK[38379] := 16#EA69;
   // UNICODE_TO_GBK[38380] := 16#9629;
   // UNICODE_TO_GBK[38381] := 16#EA6A;
   // UNICODE_TO_GBK[38382] := 16#962A;
   // UNICODE_TO_GBK[38383] := 16#DAE6;
   // UNICODE_TO_GBK[38384] := 16#962B;
   // UNICODE_TO_GBK[38385] := 16#EA6B;
   // UNICODE_TO_GBK[38386] := 16#962C;
   // UNICODE_TO_GBK[38387] := 16#EA6C;
   // UNICODE_TO_GBK[38388] := 16#962D;
   // UNICODE_TO_GBK[38389] := 16#EA6D;
   // UNICODE_TO_GBK[38390] := 16#962E;
   // UNICODE_TO_GBK[38391] := 16#C8EE;
   // UNICODE_TO_GBK[38392] := 16#962F;
   // UNICODE_TO_GBK[38393] := 16#EA6E;
   // UNICODE_TO_GBK[38394] := 16#9630;
   // UNICODE_TO_GBK[38395] := 16#EA6F;
   // UNICODE_TO_GBK[38396] := 16#9631;
   // UNICODE_TO_GBK[38397] := 16#DAE5;
   // UNICODE_TO_GBK[38398] := 16#9632;
   // UNICODE_TO_GBK[38399] := 16#B7C0;
   // UNICODE_TO_GBK[38400] := 16#9633;
   // UNICODE_TO_GBK[38401] := 16#D1F4;
   // UNICODE_TO_GBK[38402] := 16#9634;
   // UNICODE_TO_GBK[38403] := 16#D2F5;
   // UNICODE_TO_GBK[38404] := 16#9635;
   // UNICODE_TO_GBK[38405] := 16#D5F3;
   // UNICODE_TO_GBK[38406] := 16#9636;
   // UNICODE_TO_GBK[38407] := 16#BDD7;
   // UNICODE_TO_GBK[38408] := 16#9637;
   // UNICODE_TO_GBK[38409] := 16#EA70;
   // UNICODE_TO_GBK[38410] := 16#9638;
   // UNICODE_TO_GBK[38411] := 16#EA71;
   // UNICODE_TO_GBK[38412] := 16#9639;
   // UNICODE_TO_GBK[38413] := 16#EA72;
   // UNICODE_TO_GBK[38414] := 16#963A;
   // UNICODE_TO_GBK[38415] := 16#EA73;
   // UNICODE_TO_GBK[38416] := 16#963B;
   // UNICODE_TO_GBK[38417] := 16#D7E8;
   // UNICODE_TO_GBK[38418] := 16#963C;
   // UNICODE_TO_GBK[38419] := 16#DAE8;
   // UNICODE_TO_GBK[38420] := 16#963D;
   // UNICODE_TO_GBK[38421] := 16#DAE7;
   // UNICODE_TO_GBK[38422] := 16#963E;
   // UNICODE_TO_GBK[38423] := 16#EA74;
   // UNICODE_TO_GBK[38424] := 16#963F;
   // UNICODE_TO_GBK[38425] := 16#B0A2;
   // UNICODE_TO_GBK[38426] := 16#9640;
   // UNICODE_TO_GBK[38427] := 16#CDD3;
   // UNICODE_TO_GBK[38428] := 16#9641;
   // UNICODE_TO_GBK[38429] := 16#EA75;
   // UNICODE_TO_GBK[38430] := 16#9642;
   // UNICODE_TO_GBK[38431] := 16#DAE9;
   // UNICODE_TO_GBK[38432] := 16#9643;
   // UNICODE_TO_GBK[38433] := 16#EA76;
   // UNICODE_TO_GBK[38434] := 16#9644;
   // UNICODE_TO_GBK[38435] := 16#B8BD;
   // UNICODE_TO_GBK[38436] := 16#9645;
   // UNICODE_TO_GBK[38437] := 16#BCCA;
   // UNICODE_TO_GBK[38438] := 16#9646;
   // UNICODE_TO_GBK[38439] := 16#C2BD;
   // UNICODE_TO_GBK[38440] := 16#9647;
   // UNICODE_TO_GBK[38441] := 16#C2A4;
   // UNICODE_TO_GBK[38442] := 16#9648;
   // UNICODE_TO_GBK[38443] := 16#B3C2;
   // UNICODE_TO_GBK[38444] := 16#9649;
   // UNICODE_TO_GBK[38445] := 16#DAEA;
   // UNICODE_TO_GBK[38446] := 16#964A;
   // UNICODE_TO_GBK[38447] := 16#EA77;
   // UNICODE_TO_GBK[38448] := 16#964B;
   // UNICODE_TO_GBK[38449] := 16#C2AA;
   // UNICODE_TO_GBK[38450] := 16#964C;
   // UNICODE_TO_GBK[38451] := 16#C4B0;
   // UNICODE_TO_GBK[38452] := 16#964D;
   // UNICODE_TO_GBK[38453] := 16#BDB5;
   // UNICODE_TO_GBK[38454] := 16#964E;
   // UNICODE_TO_GBK[38455] := 16#EA78;
   // UNICODE_TO_GBK[38456] := 16#964F;
   // UNICODE_TO_GBK[38457] := 16#EA79;
   // UNICODE_TO_GBK[38458] := 16#9650;
   // UNICODE_TO_GBK[38459] := 16#CFDE;
   // UNICODE_TO_GBK[38460] := 16#9651;
   // UNICODE_TO_GBK[38461] := 16#EA7A;
   // UNICODE_TO_GBK[38462] := 16#9652;
   // UNICODE_TO_GBK[38463] := 16#EA7B;
   // UNICODE_TO_GBK[38464] := 16#9653;
   // UNICODE_TO_GBK[38465] := 16#EA7C;
   // UNICODE_TO_GBK[38466] := 16#9654;
   // UNICODE_TO_GBK[38467] := 16#DAEB;
   // UNICODE_TO_GBK[38468] := 16#9655;
   // UNICODE_TO_GBK[38469] := 16#C9C2;
   // UNICODE_TO_GBK[38470] := 16#9656;
   // UNICODE_TO_GBK[38471] := 16#EA7D;
   // UNICODE_TO_GBK[38472] := 16#9657;
   // UNICODE_TO_GBK[38473] := 16#EA7E;
   // UNICODE_TO_GBK[38474] := 16#9658;
   // UNICODE_TO_GBK[38475] := 16#EA80;
   // UNICODE_TO_GBK[38476] := 16#9659;
   // UNICODE_TO_GBK[38477] := 16#EA81;
   // UNICODE_TO_GBK[38478] := 16#965A;
   // UNICODE_TO_GBK[38479] := 16#EA82;
   // UNICODE_TO_GBK[38480] := 16#965B;
   // UNICODE_TO_GBK[38481] := 16#B1DD;
   // UNICODE_TO_GBK[38482] := 16#965C;
   // UNICODE_TO_GBK[38483] := 16#EA83;
   // UNICODE_TO_GBK[38484] := 16#965D;
   // UNICODE_TO_GBK[38485] := 16#EA84;
   // UNICODE_TO_GBK[38486] := 16#965E;
   // UNICODE_TO_GBK[38487] := 16#EA85;
   // UNICODE_TO_GBK[38488] := 16#965F;
   // UNICODE_TO_GBK[38489] := 16#DAEC;
   // UNICODE_TO_GBK[38490] := 16#9660;
   // UNICODE_TO_GBK[38491] := 16#EA86;
   // UNICODE_TO_GBK[38492] := 16#9661;
   // UNICODE_TO_GBK[38493] := 16#B6B8;
   // UNICODE_TO_GBK[38494] := 16#9662;
   // UNICODE_TO_GBK[38495] := 16#D4BA;
   // UNICODE_TO_GBK[38496] := 16#9663;
   // UNICODE_TO_GBK[38497] := 16#EA87;
   // UNICODE_TO_GBK[38498] := 16#9664;
   // UNICODE_TO_GBK[38499] := 16#B3FD;
   // UNICODE_TO_GBK[38500] := 16#9665;
   // UNICODE_TO_GBK[38501] := 16#EA88;
   // UNICODE_TO_GBK[38502] := 16#9666;
   // UNICODE_TO_GBK[38503] := 16#EA89;
   // UNICODE_TO_GBK[38504] := 16#9667;
   // UNICODE_TO_GBK[38505] := 16#DAED;
   // UNICODE_TO_GBK[38506] := 16#9668;
   // UNICODE_TO_GBK[38507] := 16#D4C9;
   // UNICODE_TO_GBK[38508] := 16#9669;
   // UNICODE_TO_GBK[38509] := 16#CFD5;
   // UNICODE_TO_GBK[38510] := 16#966A;
   // UNICODE_TO_GBK[38511] := 16#C5E3;
   // UNICODE_TO_GBK[38512] := 16#966B;
   // UNICODE_TO_GBK[38513] := 16#EA8A;
   // UNICODE_TO_GBK[38514] := 16#966C;
   // UNICODE_TO_GBK[38515] := 16#DAEE;
   // UNICODE_TO_GBK[38516] := 16#966D;
   // UNICODE_TO_GBK[38517] := 16#EA8B;
   // UNICODE_TO_GBK[38518] := 16#966E;
   // UNICODE_TO_GBK[38519] := 16#EA8C;
   // UNICODE_TO_GBK[38520] := 16#966F;
   // UNICODE_TO_GBK[38521] := 16#EA8D;
   // UNICODE_TO_GBK[38522] := 16#9670;
   // UNICODE_TO_GBK[38523] := 16#EA8E;
   // UNICODE_TO_GBK[38524] := 16#9671;
   // UNICODE_TO_GBK[38525] := 16#EA8F;
   // UNICODE_TO_GBK[38526] := 16#9672;
   // UNICODE_TO_GBK[38527] := 16#DAEF;
   // UNICODE_TO_GBK[38528] := 16#9673;
   // UNICODE_TO_GBK[38529] := 16#EA90;
   // UNICODE_TO_GBK[38530] := 16#9674;
   // UNICODE_TO_GBK[38531] := 16#DAF0;
   // UNICODE_TO_GBK[38532] := 16#9675;
   // UNICODE_TO_GBK[38533] := 16#C1EA;
   // UNICODE_TO_GBK[38534] := 16#9676;
   // UNICODE_TO_GBK[38535] := 16#CCD5;
   // UNICODE_TO_GBK[38536] := 16#9677;
   // UNICODE_TO_GBK[38537] := 16#CFDD;
   // UNICODE_TO_GBK[38538] := 16#9678;
   // UNICODE_TO_GBK[38539] := 16#EA91;
   // UNICODE_TO_GBK[38540] := 16#9679;
   // UNICODE_TO_GBK[38541] := 16#EA92;
   // UNICODE_TO_GBK[38542] := 16#967A;
   // UNICODE_TO_GBK[38543] := 16#EA93;
   // UNICODE_TO_GBK[38544] := 16#967B;
   // UNICODE_TO_GBK[38545] := 16#EA94;
   // UNICODE_TO_GBK[38546] := 16#967C;
   // UNICODE_TO_GBK[38547] := 16#EA95;
   // UNICODE_TO_GBK[38548] := 16#967D;
   // UNICODE_TO_GBK[38549] := 16#EA96;
   // UNICODE_TO_GBK[38550] := 16#967E;
   // UNICODE_TO_GBK[38551] := 16#EA97;
   // UNICODE_TO_GBK[38552] := 16#967F;
   // UNICODE_TO_GBK[38553] := 16#EA98;
   // UNICODE_TO_GBK[38554] := 16#9680;
   // UNICODE_TO_GBK[38555] := 16#EA99;
   // UNICODE_TO_GBK[38556] := 16#9681;
   // UNICODE_TO_GBK[38557] := 16#EA9A;
   // UNICODE_TO_GBK[38558] := 16#9682;
   // UNICODE_TO_GBK[38559] := 16#EA9B;
   // UNICODE_TO_GBK[38560] := 16#9683;
   // UNICODE_TO_GBK[38561] := 16#EA9C;
   // UNICODE_TO_GBK[38562] := 16#9684;
   // UNICODE_TO_GBK[38563] := 16#EA9D;
   // UNICODE_TO_GBK[38564] := 16#9685;
   // UNICODE_TO_GBK[38565] := 16#D3E7;
   // UNICODE_TO_GBK[38566] := 16#9686;
   // UNICODE_TO_GBK[38567] := 16#C2A1;
   // UNICODE_TO_GBK[38568] := 16#9687;
   // UNICODE_TO_GBK[38569] := 16#EA9E;
   // UNICODE_TO_GBK[38570] := 16#9688;
   // UNICODE_TO_GBK[38571] := 16#DAF1;
   // UNICODE_TO_GBK[38572] := 16#9689;
   // UNICODE_TO_GBK[38573] := 16#EA9F;
   // UNICODE_TO_GBK[38574] := 16#968A;
   // UNICODE_TO_GBK[38575] := 16#EAA0;
   // UNICODE_TO_GBK[38576] := 16#968B;
   // UNICODE_TO_GBK[38577] := 16#CBE5;
   // UNICODE_TO_GBK[38578] := 16#968C;
   // UNICODE_TO_GBK[38579] := 16#EB40;
   // UNICODE_TO_GBK[38580] := 16#968D;
   // UNICODE_TO_GBK[38581] := 16#DAF2;
   // UNICODE_TO_GBK[38582] := 16#968E;
   // UNICODE_TO_GBK[38583] := 16#EB41;
   // UNICODE_TO_GBK[38584] := 16#968F;
   // UNICODE_TO_GBK[38585] := 16#CBE6;
   // UNICODE_TO_GBK[38586] := 16#9690;
   // UNICODE_TO_GBK[38587] := 16#D2FE;
   // UNICODE_TO_GBK[38588] := 16#9691;
   // UNICODE_TO_GBK[38589] := 16#EB42;
   // UNICODE_TO_GBK[38590] := 16#9692;
   // UNICODE_TO_GBK[38591] := 16#EB43;
   // UNICODE_TO_GBK[38592] := 16#9693;
   // UNICODE_TO_GBK[38593] := 16#EB44;
   // UNICODE_TO_GBK[38594] := 16#9694;
   // UNICODE_TO_GBK[38595] := 16#B8F4;
   // UNICODE_TO_GBK[38596] := 16#9695;
   // UNICODE_TO_GBK[38597] := 16#EB45;
   // UNICODE_TO_GBK[38598] := 16#9696;
   // UNICODE_TO_GBK[38599] := 16#EB46;
   // UNICODE_TO_GBK[38600] := 16#9697;
   // UNICODE_TO_GBK[38601] := 16#DAF3;
   // UNICODE_TO_GBK[38602] := 16#9698;
   // UNICODE_TO_GBK[38603] := 16#B0AF;
   // UNICODE_TO_GBK[38604] := 16#9699;
   // UNICODE_TO_GBK[38605] := 16#CFB6;
   // UNICODE_TO_GBK[38606] := 16#969A;
   // UNICODE_TO_GBK[38607] := 16#EB47;
   // UNICODE_TO_GBK[38608] := 16#969B;
   // UNICODE_TO_GBK[38609] := 16#EB48;
   // UNICODE_TO_GBK[38610] := 16#969C;
   // UNICODE_TO_GBK[38611] := 16#D5CF;
   // UNICODE_TO_GBK[38612] := 16#969D;
   // UNICODE_TO_GBK[38613] := 16#EB49;
   // UNICODE_TO_GBK[38614] := 16#969E;
   // UNICODE_TO_GBK[38615] := 16#EB4A;
   // UNICODE_TO_GBK[38616] := 16#969F;
   // UNICODE_TO_GBK[38617] := 16#EB4B;
   // UNICODE_TO_GBK[38618] := 16#96A0;
   // UNICODE_TO_GBK[38619] := 16#EB4C;
   // UNICODE_TO_GBK[38620] := 16#96A1;
   // UNICODE_TO_GBK[38621] := 16#EB4D;
   // UNICODE_TO_GBK[38622] := 16#96A2;
   // UNICODE_TO_GBK[38623] := 16#EB4E;
   // UNICODE_TO_GBK[38624] := 16#96A3;
   // UNICODE_TO_GBK[38625] := 16#EB4F;
   // UNICODE_TO_GBK[38626] := 16#96A4;
   // UNICODE_TO_GBK[38627] := 16#EB50;
   // UNICODE_TO_GBK[38628] := 16#96A5;
   // UNICODE_TO_GBK[38629] := 16#EB51;
   // UNICODE_TO_GBK[38630] := 16#96A6;
   // UNICODE_TO_GBK[38631] := 16#EB52;
   // UNICODE_TO_GBK[38632] := 16#96A7;
   // UNICODE_TO_GBK[38633] := 16#CBED;
   // UNICODE_TO_GBK[38634] := 16#96A8;
   // UNICODE_TO_GBK[38635] := 16#EB53;
   // UNICODE_TO_GBK[38636] := 16#96A9;
   // UNICODE_TO_GBK[38637] := 16#EB54;
   // UNICODE_TO_GBK[38638] := 16#96AA;
   // UNICODE_TO_GBK[38639] := 16#EB55;
   // UNICODE_TO_GBK[38640] := 16#96AB;
   // UNICODE_TO_GBK[38641] := 16#EB56;
   // UNICODE_TO_GBK[38642] := 16#96AC;
   // UNICODE_TO_GBK[38643] := 16#EB57;
   // UNICODE_TO_GBK[38644] := 16#96AD;
   // UNICODE_TO_GBK[38645] := 16#EB58;
   // UNICODE_TO_GBK[38646] := 16#96AE;
   // UNICODE_TO_GBK[38647] := 16#EB59;
   // UNICODE_TO_GBK[38648] := 16#96AF;
   // UNICODE_TO_GBK[38649] := 16#EB5A;
   // UNICODE_TO_GBK[38650] := 16#96B0;
   // UNICODE_TO_GBK[38651] := 16#DAF4;
   // UNICODE_TO_GBK[38652] := 16#96B1;
   // UNICODE_TO_GBK[38653] := 16#EB5B;
   // UNICODE_TO_GBK[38654] := 16#96B2;
   // UNICODE_TO_GBK[38655] := 16#EB5C;
   // UNICODE_TO_GBK[38656] := 16#96B3;
   // UNICODE_TO_GBK[38657] := 16#E3C4;
   // UNICODE_TO_GBK[38658] := 16#96B4;
   // UNICODE_TO_GBK[38659] := 16#EB5D;
   // UNICODE_TO_GBK[38660] := 16#96B5;
   // UNICODE_TO_GBK[38661] := 16#EB5E;
   // UNICODE_TO_GBK[38662] := 16#96B6;
   // UNICODE_TO_GBK[38663] := 16#C1A5;
   // UNICODE_TO_GBK[38664] := 16#96B7;
   // UNICODE_TO_GBK[38665] := 16#EB5F;
   // UNICODE_TO_GBK[38666] := 16#96B8;
   // UNICODE_TO_GBK[38667] := 16#EB60;
   // UNICODE_TO_GBK[38668] := 16#96B9;
   // UNICODE_TO_GBK[38669] := 16#F6BF;
   // UNICODE_TO_GBK[38670] := 16#96BA;
   // UNICODE_TO_GBK[38671] := 16#EB61;
   // UNICODE_TO_GBK[38672] := 16#96BB;
   // UNICODE_TO_GBK[38673] := 16#EB62;
   // UNICODE_TO_GBK[38674] := 16#96BC;
   // UNICODE_TO_GBK[38675] := 16#F6C0;
   // UNICODE_TO_GBK[38676] := 16#96BD;
   // UNICODE_TO_GBK[38677] := 16#F6C1;
   // UNICODE_TO_GBK[38678] := 16#96BE;
   // UNICODE_TO_GBK[38679] := 16#C4D1;
   // UNICODE_TO_GBK[38680] := 16#96BF;
   // UNICODE_TO_GBK[38681] := 16#EB63;
   // UNICODE_TO_GBK[38682] := 16#96C0;
   // UNICODE_TO_GBK[38683] := 16#C8B8;
   // UNICODE_TO_GBK[38684] := 16#96C1;
   // UNICODE_TO_GBK[38685] := 16#D1E3;
   // UNICODE_TO_GBK[38686] := 16#96C2;
   // UNICODE_TO_GBK[38687] := 16#EB64;
   // UNICODE_TO_GBK[38688] := 16#96C3;
   // UNICODE_TO_GBK[38689] := 16#EB65;
   // UNICODE_TO_GBK[38690] := 16#96C4;
   // UNICODE_TO_GBK[38691] := 16#D0DB;
   // UNICODE_TO_GBK[38692] := 16#96C5;
   // UNICODE_TO_GBK[38693] := 16#D1C5;
   // UNICODE_TO_GBK[38694] := 16#96C6;
   // UNICODE_TO_GBK[38695] := 16#BCAF;
   // UNICODE_TO_GBK[38696] := 16#96C7;
   // UNICODE_TO_GBK[38697] := 16#B9CD;
   // UNICODE_TO_GBK[38698] := 16#96C8;
   // UNICODE_TO_GBK[38699] := 16#EB66;
   // UNICODE_TO_GBK[38700] := 16#96C9;
   // UNICODE_TO_GBK[38701] := 16#EFF4;
   // UNICODE_TO_GBK[38702] := 16#96CA;
   // UNICODE_TO_GBK[38703] := 16#EB67;
   // UNICODE_TO_GBK[38704] := 16#96CB;
   // UNICODE_TO_GBK[38705] := 16#EB68;
   // UNICODE_TO_GBK[38706] := 16#96CC;
   // UNICODE_TO_GBK[38707] := 16#B4C6;
   // UNICODE_TO_GBK[38708] := 16#96CD;
   // UNICODE_TO_GBK[38709] := 16#D3BA;
   // UNICODE_TO_GBK[38710] := 16#96CE;
   // UNICODE_TO_GBK[38711] := 16#F6C2;
   // UNICODE_TO_GBK[38712] := 16#96CF;
   // UNICODE_TO_GBK[38713] := 16#B3FB;
   // UNICODE_TO_GBK[38714] := 16#96D0;
   // UNICODE_TO_GBK[38715] := 16#EB69;
   // UNICODE_TO_GBK[38716] := 16#96D1;
   // UNICODE_TO_GBK[38717] := 16#EB6A;
   // UNICODE_TO_GBK[38718] := 16#96D2;
   // UNICODE_TO_GBK[38719] := 16#F6C3;
   // UNICODE_TO_GBK[38720] := 16#96D3;
   // UNICODE_TO_GBK[38721] := 16#EB6B;
   // UNICODE_TO_GBK[38722] := 16#96D4;
   // UNICODE_TO_GBK[38723] := 16#EB6C;
   // UNICODE_TO_GBK[38724] := 16#96D5;
   // UNICODE_TO_GBK[38725] := 16#B5F1;
   // UNICODE_TO_GBK[38726] := 16#96D6;
   // UNICODE_TO_GBK[38727] := 16#EB6D;
   // UNICODE_TO_GBK[38728] := 16#96D7;
   // UNICODE_TO_GBK[38729] := 16#EB6E;
   // UNICODE_TO_GBK[38730] := 16#96D8;
   // UNICODE_TO_GBK[38731] := 16#EB6F;
   // UNICODE_TO_GBK[38732] := 16#96D9;
   // UNICODE_TO_GBK[38733] := 16#EB70;
   // UNICODE_TO_GBK[38734] := 16#96DA;
   // UNICODE_TO_GBK[38735] := 16#EB71;
   // UNICODE_TO_GBK[38736] := 16#96DB;
   // UNICODE_TO_GBK[38737] := 16#EB72;
   // UNICODE_TO_GBK[38738] := 16#96DC;
   // UNICODE_TO_GBK[38739] := 16#EB73;
   // UNICODE_TO_GBK[38740] := 16#96DD;
   // UNICODE_TO_GBK[38741] := 16#EB74;
   // UNICODE_TO_GBK[38742] := 16#96DE;
   // UNICODE_TO_GBK[38743] := 16#EB75;
   // UNICODE_TO_GBK[38744] := 16#96DF;
   // UNICODE_TO_GBK[38745] := 16#EB76;
   // UNICODE_TO_GBK[38746] := 16#96E0;
   // UNICODE_TO_GBK[38747] := 16#F6C5;
   // UNICODE_TO_GBK[38748] := 16#96E1;
   // UNICODE_TO_GBK[38749] := 16#EB77;
   // UNICODE_TO_GBK[38750] := 16#96E2;
   // UNICODE_TO_GBK[38751] := 16#EB78;
   // UNICODE_TO_GBK[38752] := 16#96E3;
   // UNICODE_TO_GBK[38753] := 16#EB79;
   // UNICODE_TO_GBK[38754] := 16#96E4;
   // UNICODE_TO_GBK[38755] := 16#EB7A;
   // UNICODE_TO_GBK[38756] := 16#96E5;
   // UNICODE_TO_GBK[38757] := 16#EB7B;
   // UNICODE_TO_GBK[38758] := 16#96E6;
   // UNICODE_TO_GBK[38759] := 16#EB7C;
   // UNICODE_TO_GBK[38760] := 16#96E7;
   // UNICODE_TO_GBK[38761] := 16#EB7D;
   // UNICODE_TO_GBK[38762] := 16#96E8;
   // UNICODE_TO_GBK[38763] := 16#D3EA;
   // UNICODE_TO_GBK[38764] := 16#96E9;
   // UNICODE_TO_GBK[38765] := 16#F6A7;
   // UNICODE_TO_GBK[38766] := 16#96EA;
   // UNICODE_TO_GBK[38767] := 16#D1A9;
   // UNICODE_TO_GBK[38768] := 16#96EB;
   // UNICODE_TO_GBK[38769] := 16#EB7E;
   // UNICODE_TO_GBK[38770] := 16#96EC;
   // UNICODE_TO_GBK[38771] := 16#EB80;
   // UNICODE_TO_GBK[38772] := 16#96ED;
   // UNICODE_TO_GBK[38773] := 16#EB81;
   // UNICODE_TO_GBK[38774] := 16#96EE;
   // UNICODE_TO_GBK[38775] := 16#EB82;
   // UNICODE_TO_GBK[38776] := 16#96EF;
   // UNICODE_TO_GBK[38777] := 16#F6A9;
   // UNICODE_TO_GBK[38778] := 16#96F0;
   // UNICODE_TO_GBK[38779] := 16#EB83;
   // UNICODE_TO_GBK[38780] := 16#96F1;
   // UNICODE_TO_GBK[38781] := 16#EB84;
   // UNICODE_TO_GBK[38782] := 16#96F2;
   // UNICODE_TO_GBK[38783] := 16#EB85;
   // UNICODE_TO_GBK[38784] := 16#96F3;
   // UNICODE_TO_GBK[38785] := 16#F6A8;
   // UNICODE_TO_GBK[38786] := 16#96F4;
   // UNICODE_TO_GBK[38787] := 16#EB86;
   // UNICODE_TO_GBK[38788] := 16#96F5;
   // UNICODE_TO_GBK[38789] := 16#EB87;
   // UNICODE_TO_GBK[38790] := 16#96F6;
   // UNICODE_TO_GBK[38791] := 16#C1E3;
   // UNICODE_TO_GBK[38792] := 16#96F7;
   // UNICODE_TO_GBK[38793] := 16#C0D7;
   // UNICODE_TO_GBK[38794] := 16#96F8;
   // UNICODE_TO_GBK[38795] := 16#EB88;
   // UNICODE_TO_GBK[38796] := 16#96F9;
   // UNICODE_TO_GBK[38797] := 16#B1A2;
   // UNICODE_TO_GBK[38798] := 16#96FA;
   // UNICODE_TO_GBK[38799] := 16#EB89;
   // UNICODE_TO_GBK[38800] := 16#96FB;
   // UNICODE_TO_GBK[38801] := 16#EB8A;
   // UNICODE_TO_GBK[38802] := 16#96FC;
   // UNICODE_TO_GBK[38803] := 16#EB8B;
   // UNICODE_TO_GBK[38804] := 16#96FD;
   // UNICODE_TO_GBK[38805] := 16#EB8C;
   // UNICODE_TO_GBK[38806] := 16#96FE;
   // UNICODE_TO_GBK[38807] := 16#CEED;
   // UNICODE_TO_GBK[38808] := 16#96FF;
   // UNICODE_TO_GBK[38809] := 16#EB8D;
   // UNICODE_TO_GBK[38810] := 16#9700;
   // UNICODE_TO_GBK[38811] := 16#D0E8;
   // UNICODE_TO_GBK[38812] := 16#9701;
   // UNICODE_TO_GBK[38813] := 16#F6AB;
   // UNICODE_TO_GBK[38814] := 16#9702;
   // UNICODE_TO_GBK[38815] := 16#EB8E;
   // UNICODE_TO_GBK[38816] := 16#9703;
   // UNICODE_TO_GBK[38817] := 16#EB8F;
   // UNICODE_TO_GBK[38818] := 16#9704;
   // UNICODE_TO_GBK[38819] := 16#CFF6;
   // UNICODE_TO_GBK[38820] := 16#9705;
   // UNICODE_TO_GBK[38821] := 16#EB90;
   // UNICODE_TO_GBK[38822] := 16#9706;
   // UNICODE_TO_GBK[38823] := 16#F6AA;
   // UNICODE_TO_GBK[38824] := 16#9707;
   // UNICODE_TO_GBK[38825] := 16#D5F0;
   // UNICODE_TO_GBK[38826] := 16#9708;
   // UNICODE_TO_GBK[38827] := 16#F6AC;
   // UNICODE_TO_GBK[38828] := 16#9709;
   // UNICODE_TO_GBK[38829] := 16#C3B9;
   // UNICODE_TO_GBK[38830] := 16#970A;
   // UNICODE_TO_GBK[38831] := 16#EB91;
   // UNICODE_TO_GBK[38832] := 16#970B;
   // UNICODE_TO_GBK[38833] := 16#EB92;
   // UNICODE_TO_GBK[38834] := 16#970C;
   // UNICODE_TO_GBK[38835] := 16#EB93;
   // UNICODE_TO_GBK[38836] := 16#970D;
   // UNICODE_TO_GBK[38837] := 16#BBF4;
   // UNICODE_TO_GBK[38838] := 16#970E;
   // UNICODE_TO_GBK[38839] := 16#F6AE;
   // UNICODE_TO_GBK[38840] := 16#970F;
   // UNICODE_TO_GBK[38841] := 16#F6AD;
   // UNICODE_TO_GBK[38842] := 16#9710;
   // UNICODE_TO_GBK[38843] := 16#EB94;
   // UNICODE_TO_GBK[38844] := 16#9711;
   // UNICODE_TO_GBK[38845] := 16#EB95;
   // UNICODE_TO_GBK[38846] := 16#9712;
   // UNICODE_TO_GBK[38847] := 16#EB96;
   // UNICODE_TO_GBK[38848] := 16#9713;
   // UNICODE_TO_GBK[38849] := 16#C4DE;
   // UNICODE_TO_GBK[38850] := 16#9714;
   // UNICODE_TO_GBK[38851] := 16#EB97;
   // UNICODE_TO_GBK[38852] := 16#9715;
   // UNICODE_TO_GBK[38853] := 16#EB98;
   // UNICODE_TO_GBK[38854] := 16#9716;
   // UNICODE_TO_GBK[38855] := 16#C1D8;
   // UNICODE_TO_GBK[38856] := 16#9717;
   // UNICODE_TO_GBK[38857] := 16#EB99;
   // UNICODE_TO_GBK[38858] := 16#9718;
   // UNICODE_TO_GBK[38859] := 16#EB9A;
   // UNICODE_TO_GBK[38860] := 16#9719;
   // UNICODE_TO_GBK[38861] := 16#EB9B;
   // UNICODE_TO_GBK[38862] := 16#971A;
   // UNICODE_TO_GBK[38863] := 16#EB9C;
   // UNICODE_TO_GBK[38864] := 16#971B;
   // UNICODE_TO_GBK[38865] := 16#EB9D;
   // UNICODE_TO_GBK[38866] := 16#971C;
   // UNICODE_TO_GBK[38867] := 16#CBAA;
   // UNICODE_TO_GBK[38868] := 16#971D;
   // UNICODE_TO_GBK[38869] := 16#EB9E;
   // UNICODE_TO_GBK[38870] := 16#971E;
   // UNICODE_TO_GBK[38871] := 16#CFBC;
   // UNICODE_TO_GBK[38872] := 16#971F;
   // UNICODE_TO_GBK[38873] := 16#EB9F;
   // UNICODE_TO_GBK[38874] := 16#9720;
   // UNICODE_TO_GBK[38875] := 16#EBA0;
   // UNICODE_TO_GBK[38876] := 16#9721;
   // UNICODE_TO_GBK[38877] := 16#EC40;
   // UNICODE_TO_GBK[38878] := 16#9722;
   // UNICODE_TO_GBK[38879] := 16#EC41;
   // UNICODE_TO_GBK[38880] := 16#9723;
   // UNICODE_TO_GBK[38881] := 16#EC42;
   // UNICODE_TO_GBK[38882] := 16#9724;
   // UNICODE_TO_GBK[38883] := 16#EC43;
   // UNICODE_TO_GBK[38884] := 16#9725;
   // UNICODE_TO_GBK[38885] := 16#EC44;
   // UNICODE_TO_GBK[38886] := 16#9726;
   // UNICODE_TO_GBK[38887] := 16#EC45;
   // UNICODE_TO_GBK[38888] := 16#9727;
   // UNICODE_TO_GBK[38889] := 16#EC46;
   // UNICODE_TO_GBK[38890] := 16#9728;
   // UNICODE_TO_GBK[38891] := 16#EC47;
   // UNICODE_TO_GBK[38892] := 16#9729;
   // UNICODE_TO_GBK[38893] := 16#EC48;
   // UNICODE_TO_GBK[38894] := 16#972A;
   // UNICODE_TO_GBK[38895] := 16#F6AF;
   // UNICODE_TO_GBK[38896] := 16#972B;
   // UNICODE_TO_GBK[38897] := 16#EC49;
   // UNICODE_TO_GBK[38898] := 16#972C;
   // UNICODE_TO_GBK[38899] := 16#EC4A;
   // UNICODE_TO_GBK[38900] := 16#972D;
   // UNICODE_TO_GBK[38901] := 16#F6B0;
   // UNICODE_TO_GBK[38902] := 16#972E;
   // UNICODE_TO_GBK[38903] := 16#EC4B;
   // UNICODE_TO_GBK[38904] := 16#972F;
   // UNICODE_TO_GBK[38905] := 16#EC4C;
   // UNICODE_TO_GBK[38906] := 16#9730;
   // UNICODE_TO_GBK[38907] := 16#F6B1;
   // UNICODE_TO_GBK[38908] := 16#9731;
   // UNICODE_TO_GBK[38909] := 16#EC4D;
   // UNICODE_TO_GBK[38910] := 16#9732;
   // UNICODE_TO_GBK[38911] := 16#C2B6;
   // UNICODE_TO_GBK[38912] := 16#9733;
   // UNICODE_TO_GBK[38913] := 16#EC4E;
   // UNICODE_TO_GBK[38914] := 16#9734;
   // UNICODE_TO_GBK[38915] := 16#EC4F;
   // UNICODE_TO_GBK[38916] := 16#9735;
   // UNICODE_TO_GBK[38917] := 16#EC50;
   // UNICODE_TO_GBK[38918] := 16#9736;
   // UNICODE_TO_GBK[38919] := 16#EC51;
   // UNICODE_TO_GBK[38920] := 16#9737;
   // UNICODE_TO_GBK[38921] := 16#EC52;
   // UNICODE_TO_GBK[38922] := 16#9738;
   // UNICODE_TO_GBK[38923] := 16#B0D4;
   // UNICODE_TO_GBK[38924] := 16#9739;
   // UNICODE_TO_GBK[38925] := 16#C5F9;
   // UNICODE_TO_GBK[38926] := 16#973A;
   // UNICODE_TO_GBK[38927] := 16#EC53;
   // UNICODE_TO_GBK[38928] := 16#973B;
   // UNICODE_TO_GBK[38929] := 16#EC54;
   // UNICODE_TO_GBK[38930] := 16#973C;
   // UNICODE_TO_GBK[38931] := 16#EC55;
   // UNICODE_TO_GBK[38932] := 16#973D;
   // UNICODE_TO_GBK[38933] := 16#EC56;
   // UNICODE_TO_GBK[38934] := 16#973E;
   // UNICODE_TO_GBK[38935] := 16#F6B2;
   // UNICODE_TO_GBK[38936] := 16#973F;
   // UNICODE_TO_GBK[38937] := 16#EC57;
   // UNICODE_TO_GBK[38938] := 16#9740;
   // UNICODE_TO_GBK[38939] := 16#EC58;
   // UNICODE_TO_GBK[38940] := 16#9741;
   // UNICODE_TO_GBK[38941] := 16#EC59;
   // UNICODE_TO_GBK[38942] := 16#9742;
   // UNICODE_TO_GBK[38943] := 16#EC5A;
   // UNICODE_TO_GBK[38944] := 16#9743;
   // UNICODE_TO_GBK[38945] := 16#EC5B;
   // UNICODE_TO_GBK[38946] := 16#9744;
   // UNICODE_TO_GBK[38947] := 16#EC5C;
   // UNICODE_TO_GBK[38948] := 16#9745;
   // UNICODE_TO_GBK[38949] := 16#EC5D;
   // UNICODE_TO_GBK[38950] := 16#9746;
   // UNICODE_TO_GBK[38951] := 16#EC5E;
   // UNICODE_TO_GBK[38952] := 16#9747;
   // UNICODE_TO_GBK[38953] := 16#EC5F;
   // UNICODE_TO_GBK[38954] := 16#9748;
   // UNICODE_TO_GBK[38955] := 16#EC60;
   // UNICODE_TO_GBK[38956] := 16#9749;
   // UNICODE_TO_GBK[38957] := 16#EC61;
   // UNICODE_TO_GBK[38958] := 16#974A;
   // UNICODE_TO_GBK[38959] := 16#EC62;
   // UNICODE_TO_GBK[38960] := 16#974B;
   // UNICODE_TO_GBK[38961] := 16#EC63;
   // UNICODE_TO_GBK[38962] := 16#974C;
   // UNICODE_TO_GBK[38963] := 16#EC64;
   // UNICODE_TO_GBK[38964] := 16#974D;
   // UNICODE_TO_GBK[38965] := 16#EC65;
   // UNICODE_TO_GBK[38966] := 16#974E;
   // UNICODE_TO_GBK[38967] := 16#EC66;
   // UNICODE_TO_GBK[38968] := 16#974F;
   // UNICODE_TO_GBK[38969] := 16#EC67;
   // UNICODE_TO_GBK[38970] := 16#9750;
   // UNICODE_TO_GBK[38971] := 16#EC68;
   // UNICODE_TO_GBK[38972] := 16#9751;
   // UNICODE_TO_GBK[38973] := 16#EC69;
   // UNICODE_TO_GBK[38974] := 16#9752;
   // UNICODE_TO_GBK[38975] := 16#C7E0;
   // UNICODE_TO_GBK[38976] := 16#9753;
   // UNICODE_TO_GBK[38977] := 16#F6A6;
   // UNICODE_TO_GBK[38978] := 16#9754;
   // UNICODE_TO_GBK[38979] := 16#EC6A;
   // UNICODE_TO_GBK[38980] := 16#9755;
   // UNICODE_TO_GBK[38981] := 16#EC6B;
   // UNICODE_TO_GBK[38982] := 16#9756;
   // UNICODE_TO_GBK[38983] := 16#BEB8;
   // UNICODE_TO_GBK[38984] := 16#9757;
   // UNICODE_TO_GBK[38985] := 16#EC6C;
   // UNICODE_TO_GBK[38986] := 16#9758;
   // UNICODE_TO_GBK[38987] := 16#EC6D;
   // UNICODE_TO_GBK[38988] := 16#9759;
   // UNICODE_TO_GBK[38989] := 16#BEB2;
   // UNICODE_TO_GBK[38990] := 16#975A;
   // UNICODE_TO_GBK[38991] := 16#EC6E;
   // UNICODE_TO_GBK[38992] := 16#975B;
   // UNICODE_TO_GBK[38993] := 16#B5E5;
   // UNICODE_TO_GBK[38994] := 16#975C;
   // UNICODE_TO_GBK[38995] := 16#EC6F;
   // UNICODE_TO_GBK[38996] := 16#975D;
   // UNICODE_TO_GBK[38997] := 16#EC70;
   // UNICODE_TO_GBK[38998] := 16#975E;
   // UNICODE_TO_GBK[38999] := 16#B7C7;
   // UNICODE_TO_GBK[39000] := 16#975F;
   // UNICODE_TO_GBK[39001] := 16#EC71;
   // UNICODE_TO_GBK[39002] := 16#9760;
   // UNICODE_TO_GBK[39003] := 16#BFBF;
   // UNICODE_TO_GBK[39004] := 16#9761;
   // UNICODE_TO_GBK[39005] := 16#C3D2;
   // UNICODE_TO_GBK[39006] := 16#9762;
   // UNICODE_TO_GBK[39007] := 16#C3E6;
   // UNICODE_TO_GBK[39008] := 16#9763;
   // UNICODE_TO_GBK[39009] := 16#EC72;
   // UNICODE_TO_GBK[39010] := 16#9764;
   // UNICODE_TO_GBK[39011] := 16#EC73;
   // UNICODE_TO_GBK[39012] := 16#9765;
   // UNICODE_TO_GBK[39013] := 16#D8CC;
   // UNICODE_TO_GBK[39014] := 16#9766;
   // UNICODE_TO_GBK[39015] := 16#EC74;
   // UNICODE_TO_GBK[39016] := 16#9767;
   // UNICODE_TO_GBK[39017] := 16#EC75;
   // UNICODE_TO_GBK[39018] := 16#9768;
   // UNICODE_TO_GBK[39019] := 16#EC76;
   // UNICODE_TO_GBK[39020] := 16#9769;
   // UNICODE_TO_GBK[39021] := 16#B8EF;
   // UNICODE_TO_GBK[39022] := 16#976A;
   // UNICODE_TO_GBK[39023] := 16#EC77;
   // UNICODE_TO_GBK[39024] := 16#976B;
   // UNICODE_TO_GBK[39025] := 16#EC78;
   // UNICODE_TO_GBK[39026] := 16#976C;
   // UNICODE_TO_GBK[39027] := 16#EC79;
   // UNICODE_TO_GBK[39028] := 16#976D;
   // UNICODE_TO_GBK[39029] := 16#EC7A;
   // UNICODE_TO_GBK[39030] := 16#976E;
   // UNICODE_TO_GBK[39031] := 16#EC7B;
   // UNICODE_TO_GBK[39032] := 16#976F;
   // UNICODE_TO_GBK[39033] := 16#EC7C;
   // UNICODE_TO_GBK[39034] := 16#9770;
   // UNICODE_TO_GBK[39035] := 16#EC7D;
   // UNICODE_TO_GBK[39036] := 16#9771;
   // UNICODE_TO_GBK[39037] := 16#EC7E;
   // UNICODE_TO_GBK[39038] := 16#9772;
   // UNICODE_TO_GBK[39039] := 16#EC80;
   // UNICODE_TO_GBK[39040] := 16#9773;
   // UNICODE_TO_GBK[39041] := 16#BDF9;
   // UNICODE_TO_GBK[39042] := 16#9774;
   // UNICODE_TO_GBK[39043] := 16#D1A5;
   // UNICODE_TO_GBK[39044] := 16#9775;
   // UNICODE_TO_GBK[39045] := 16#EC81;
   // UNICODE_TO_GBK[39046] := 16#9776;
   // UNICODE_TO_GBK[39047] := 16#B0D0;
   // UNICODE_TO_GBK[39048] := 16#9777;
   // UNICODE_TO_GBK[39049] := 16#EC82;
   // UNICODE_TO_GBK[39050] := 16#9778;
   // UNICODE_TO_GBK[39051] := 16#EC83;
   // UNICODE_TO_GBK[39052] := 16#9779;
   // UNICODE_TO_GBK[39053] := 16#EC84;
   // UNICODE_TO_GBK[39054] := 16#977A;
   // UNICODE_TO_GBK[39055] := 16#EC85;
   // UNICODE_TO_GBK[39056] := 16#977B;
   // UNICODE_TO_GBK[39057] := 16#EC86;
   // UNICODE_TO_GBK[39058] := 16#977C;
   // UNICODE_TO_GBK[39059] := 16#F7B0;
   // UNICODE_TO_GBK[39060] := 16#977D;
   // UNICODE_TO_GBK[39061] := 16#EC87;
   // UNICODE_TO_GBK[39062] := 16#977E;
   // UNICODE_TO_GBK[39063] := 16#EC88;
   // UNICODE_TO_GBK[39064] := 16#977F;
   // UNICODE_TO_GBK[39065] := 16#EC89;
   // UNICODE_TO_GBK[39066] := 16#9780;
   // UNICODE_TO_GBK[39067] := 16#EC8A;
   // UNICODE_TO_GBK[39068] := 16#9781;
   // UNICODE_TO_GBK[39069] := 16#EC8B;
   // UNICODE_TO_GBK[39070] := 16#9782;
   // UNICODE_TO_GBK[39071] := 16#EC8C;
   // UNICODE_TO_GBK[39072] := 16#9783;
   // UNICODE_TO_GBK[39073] := 16#EC8D;
   // UNICODE_TO_GBK[39074] := 16#9784;
   // UNICODE_TO_GBK[39075] := 16#EC8E;
   // UNICODE_TO_GBK[39076] := 16#9785;
   // UNICODE_TO_GBK[39077] := 16#F7B1;
   // UNICODE_TO_GBK[39078] := 16#9786;
   // UNICODE_TO_GBK[39079] := 16#EC8F;
   // UNICODE_TO_GBK[39080] := 16#9787;
   // UNICODE_TO_GBK[39081] := 16#EC90;
   // UNICODE_TO_GBK[39082] := 16#9788;
   // UNICODE_TO_GBK[39083] := 16#EC91;
   // UNICODE_TO_GBK[39084] := 16#9789;
   // UNICODE_TO_GBK[39085] := 16#EC92;
   // UNICODE_TO_GBK[39086] := 16#978A;
   // UNICODE_TO_GBK[39087] := 16#EC93;
   // UNICODE_TO_GBK[39088] := 16#978B;
   // UNICODE_TO_GBK[39089] := 16#D0AC;
   // UNICODE_TO_GBK[39090] := 16#978C;
   // UNICODE_TO_GBK[39091] := 16#EC94;
   // UNICODE_TO_GBK[39092] := 16#978D;
   // UNICODE_TO_GBK[39093] := 16#B0B0;
   // UNICODE_TO_GBK[39094] := 16#978E;
   // UNICODE_TO_GBK[39095] := 16#EC95;
   // UNICODE_TO_GBK[39096] := 16#978F;
   // UNICODE_TO_GBK[39097] := 16#EC96;
   // UNICODE_TO_GBK[39098] := 16#9790;
   // UNICODE_TO_GBK[39099] := 16#EC97;
   // UNICODE_TO_GBK[39100] := 16#9791;
   // UNICODE_TO_GBK[39101] := 16#F7B2;
   // UNICODE_TO_GBK[39102] := 16#9792;
   // UNICODE_TO_GBK[39103] := 16#F7B3;
   // UNICODE_TO_GBK[39104] := 16#9793;
   // UNICODE_TO_GBK[39105] := 16#EC98;
   // UNICODE_TO_GBK[39106] := 16#9794;
   // UNICODE_TO_GBK[39107] := 16#F7B4;
   // UNICODE_TO_GBK[39108] := 16#9795;
   // UNICODE_TO_GBK[39109] := 16#EC99;
   // UNICODE_TO_GBK[39110] := 16#9796;
   // UNICODE_TO_GBK[39111] := 16#EC9A;
   // UNICODE_TO_GBK[39112] := 16#9797;
   // UNICODE_TO_GBK[39113] := 16#EC9B;
   // UNICODE_TO_GBK[39114] := 16#9798;
   // UNICODE_TO_GBK[39115] := 16#C7CA;
   // UNICODE_TO_GBK[39116] := 16#9799;
   // UNICODE_TO_GBK[39117] := 16#EC9C;
   // UNICODE_TO_GBK[39118] := 16#979A;
   // UNICODE_TO_GBK[39119] := 16#EC9D;
   // UNICODE_TO_GBK[39120] := 16#979B;
   // UNICODE_TO_GBK[39121] := 16#EC9E;
   // UNICODE_TO_GBK[39122] := 16#979C;
   // UNICODE_TO_GBK[39123] := 16#EC9F;
   // UNICODE_TO_GBK[39124] := 16#979D;
   // UNICODE_TO_GBK[39125] := 16#ECA0;
   // UNICODE_TO_GBK[39126] := 16#979E;
   // UNICODE_TO_GBK[39127] := 16#ED40;
   // UNICODE_TO_GBK[39128] := 16#979F;
   // UNICODE_TO_GBK[39129] := 16#ED41;
   // UNICODE_TO_GBK[39130] := 16#97A0;
   // UNICODE_TO_GBK[39131] := 16#BECF;
   // UNICODE_TO_GBK[39132] := 16#97A1;
   // UNICODE_TO_GBK[39133] := 16#ED42;
   // UNICODE_TO_GBK[39134] := 16#97A2;
   // UNICODE_TO_GBK[39135] := 16#ED43;
   // UNICODE_TO_GBK[39136] := 16#97A3;
   // UNICODE_TO_GBK[39137] := 16#F7B7;
   // UNICODE_TO_GBK[39138] := 16#97A4;
   // UNICODE_TO_GBK[39139] := 16#ED44;
   // UNICODE_TO_GBK[39140] := 16#97A5;
   // UNICODE_TO_GBK[39141] := 16#ED45;
   // UNICODE_TO_GBK[39142] := 16#97A6;
   // UNICODE_TO_GBK[39143] := 16#ED46;
   // UNICODE_TO_GBK[39144] := 16#97A7;
   // UNICODE_TO_GBK[39145] := 16#ED47;
   // UNICODE_TO_GBK[39146] := 16#97A8;
   // UNICODE_TO_GBK[39147] := 16#ED48;
   // UNICODE_TO_GBK[39148] := 16#97A9;
   // UNICODE_TO_GBK[39149] := 16#ED49;
   // UNICODE_TO_GBK[39150] := 16#97AA;
   // UNICODE_TO_GBK[39151] := 16#ED4A;
   // UNICODE_TO_GBK[39152] := 16#97AB;
   // UNICODE_TO_GBK[39153] := 16#F7B6;
   // UNICODE_TO_GBK[39154] := 16#97AC;
   // UNICODE_TO_GBK[39155] := 16#ED4B;
   // UNICODE_TO_GBK[39156] := 16#97AD;
   // UNICODE_TO_GBK[39157] := 16#B1DE;
   // UNICODE_TO_GBK[39158] := 16#97AE;
   // UNICODE_TO_GBK[39159] := 16#ED4C;
   // UNICODE_TO_GBK[39160] := 16#97AF;
   // UNICODE_TO_GBK[39161] := 16#F7B5;
   // UNICODE_TO_GBK[39162] := 16#97B0;
   // UNICODE_TO_GBK[39163] := 16#ED4D;
   // UNICODE_TO_GBK[39164] := 16#97B1;
   // UNICODE_TO_GBK[39165] := 16#ED4E;
   // UNICODE_TO_GBK[39166] := 16#97B2;
   // UNICODE_TO_GBK[39167] := 16#F7B8;
   // UNICODE_TO_GBK[39168] := 16#97B3;
   // UNICODE_TO_GBK[39169] := 16#ED4F;
   // UNICODE_TO_GBK[39170] := 16#97B4;
   // UNICODE_TO_GBK[39171] := 16#F7B9;
   // UNICODE_TO_GBK[39172] := 16#97B5;
   // UNICODE_TO_GBK[39173] := 16#ED50;
   // UNICODE_TO_GBK[39174] := 16#97B6;
   // UNICODE_TO_GBK[39175] := 16#ED51;
   // UNICODE_TO_GBK[39176] := 16#97B7;
   // UNICODE_TO_GBK[39177] := 16#ED52;
   // UNICODE_TO_GBK[39178] := 16#97B8;
   // UNICODE_TO_GBK[39179] := 16#ED53;
   // UNICODE_TO_GBK[39180] := 16#97B9;
   // UNICODE_TO_GBK[39181] := 16#ED54;
   // UNICODE_TO_GBK[39182] := 16#97BA;
   // UNICODE_TO_GBK[39183] := 16#ED55;
   // UNICODE_TO_GBK[39184] := 16#97BB;
   // UNICODE_TO_GBK[39185] := 16#ED56;
   // UNICODE_TO_GBK[39186] := 16#97BC;
   // UNICODE_TO_GBK[39187] := 16#ED57;
   // UNICODE_TO_GBK[39188] := 16#97BD;
   // UNICODE_TO_GBK[39189] := 16#ED58;
   // UNICODE_TO_GBK[39190] := 16#97BE;
   // UNICODE_TO_GBK[39191] := 16#ED59;
   // UNICODE_TO_GBK[39192] := 16#97BF;
   // UNICODE_TO_GBK[39193] := 16#ED5A;
   // UNICODE_TO_GBK[39194] := 16#97C0;
   // UNICODE_TO_GBK[39195] := 16#ED5B;
   // UNICODE_TO_GBK[39196] := 16#97C1;
   // UNICODE_TO_GBK[39197] := 16#ED5C;
   // UNICODE_TO_GBK[39198] := 16#97C2;
   // UNICODE_TO_GBK[39199] := 16#ED5D;
   // UNICODE_TO_GBK[39200] := 16#97C3;
   // UNICODE_TO_GBK[39201] := 16#ED5E;
   // UNICODE_TO_GBK[39202] := 16#97C4;
   // UNICODE_TO_GBK[39203] := 16#ED5F;
   // UNICODE_TO_GBK[39204] := 16#97C5;
   // UNICODE_TO_GBK[39205] := 16#ED60;
   // UNICODE_TO_GBK[39206] := 16#97C6;
   // UNICODE_TO_GBK[39207] := 16#ED61;
   // UNICODE_TO_GBK[39208] := 16#97C7;
   // UNICODE_TO_GBK[39209] := 16#ED62;
   // UNICODE_TO_GBK[39210] := 16#97C8;
   // UNICODE_TO_GBK[39211] := 16#ED63;
   // UNICODE_TO_GBK[39212] := 16#97C9;
   // UNICODE_TO_GBK[39213] := 16#ED64;
   // UNICODE_TO_GBK[39214] := 16#97CA;
   // UNICODE_TO_GBK[39215] := 16#ED65;
   // UNICODE_TO_GBK[39216] := 16#97CB;
   // UNICODE_TO_GBK[39217] := 16#ED66;
   // UNICODE_TO_GBK[39218] := 16#97CC;
   // UNICODE_TO_GBK[39219] := 16#ED67;
   // UNICODE_TO_GBK[39220] := 16#97CD;
   // UNICODE_TO_GBK[39221] := 16#ED68;
   // UNICODE_TO_GBK[39222] := 16#97CE;
   // UNICODE_TO_GBK[39223] := 16#ED69;
   // UNICODE_TO_GBK[39224] := 16#97CF;
   // UNICODE_TO_GBK[39225] := 16#ED6A;
   // UNICODE_TO_GBK[39226] := 16#97D0;
   // UNICODE_TO_GBK[39227] := 16#ED6B;
   // UNICODE_TO_GBK[39228] := 16#97D1;
   // UNICODE_TO_GBK[39229] := 16#ED6C;
   // UNICODE_TO_GBK[39230] := 16#97D2;
   // UNICODE_TO_GBK[39231] := 16#ED6D;
   // UNICODE_TO_GBK[39232] := 16#97D3;
   // UNICODE_TO_GBK[39233] := 16#ED6E;
   // UNICODE_TO_GBK[39234] := 16#97D4;
   // UNICODE_TO_GBK[39235] := 16#ED6F;
   // UNICODE_TO_GBK[39236] := 16#97D5;
   // UNICODE_TO_GBK[39237] := 16#ED70;
   // UNICODE_TO_GBK[39238] := 16#97D6;
   // UNICODE_TO_GBK[39239] := 16#ED71;
   // UNICODE_TO_GBK[39240] := 16#97D7;
   // UNICODE_TO_GBK[39241] := 16#ED72;
   // UNICODE_TO_GBK[39242] := 16#97D8;
   // UNICODE_TO_GBK[39243] := 16#ED73;
   // UNICODE_TO_GBK[39244] := 16#97D9;
   // UNICODE_TO_GBK[39245] := 16#ED74;
   // UNICODE_TO_GBK[39246] := 16#97DA;
   // UNICODE_TO_GBK[39247] := 16#ED75;
   // UNICODE_TO_GBK[39248] := 16#97DB;
   // UNICODE_TO_GBK[39249] := 16#ED76;
   // UNICODE_TO_GBK[39250] := 16#97DC;
   // UNICODE_TO_GBK[39251] := 16#ED77;
   // UNICODE_TO_GBK[39252] := 16#97DD;
   // UNICODE_TO_GBK[39253] := 16#ED78;
   // UNICODE_TO_GBK[39254] := 16#97DE;
   // UNICODE_TO_GBK[39255] := 16#ED79;
   // UNICODE_TO_GBK[39256] := 16#97DF;
   // UNICODE_TO_GBK[39257] := 16#ED7A;
   // UNICODE_TO_GBK[39258] := 16#97E0;
   // UNICODE_TO_GBK[39259] := 16#ED7B;
   // UNICODE_TO_GBK[39260] := 16#97E1;
   // UNICODE_TO_GBK[39261] := 16#ED7C;
   // UNICODE_TO_GBK[39262] := 16#97E2;
   // UNICODE_TO_GBK[39263] := 16#ED7D;
   // UNICODE_TO_GBK[39264] := 16#97E3;
   // UNICODE_TO_GBK[39265] := 16#ED7E;
   // UNICODE_TO_GBK[39266] := 16#97E4;
   // UNICODE_TO_GBK[39267] := 16#ED80;
   // UNICODE_TO_GBK[39268] := 16#97E5;
   // UNICODE_TO_GBK[39269] := 16#ED81;
   // UNICODE_TO_GBK[39270] := 16#97E6;
   // UNICODE_TO_GBK[39271] := 16#CEA4;
   // UNICODE_TO_GBK[39272] := 16#97E7;
   // UNICODE_TO_GBK[39273] := 16#C8CD;
   // UNICODE_TO_GBK[39274] := 16#97E8;
   // UNICODE_TO_GBK[39275] := 16#ED82;
   // UNICODE_TO_GBK[39276] := 16#97E9;
   // UNICODE_TO_GBK[39277] := 16#BAAB;
   // UNICODE_TO_GBK[39278] := 16#97EA;
   // UNICODE_TO_GBK[39279] := 16#E8B8;
   // UNICODE_TO_GBK[39280] := 16#97EB;
   // UNICODE_TO_GBK[39281] := 16#E8B9;
   // UNICODE_TO_GBK[39282] := 16#97EC;
   // UNICODE_TO_GBK[39283] := 16#E8BA;
   // UNICODE_TO_GBK[39284] := 16#97ED;
   // UNICODE_TO_GBK[39285] := 16#BEC2;
   // UNICODE_TO_GBK[39286] := 16#97EE;
   // UNICODE_TO_GBK[39287] := 16#ED83;
   // UNICODE_TO_GBK[39288] := 16#97EF;
   // UNICODE_TO_GBK[39289] := 16#ED84;
   // UNICODE_TO_GBK[39290] := 16#97F0;
   // UNICODE_TO_GBK[39291] := 16#ED85;
   // UNICODE_TO_GBK[39292] := 16#97F1;
   // UNICODE_TO_GBK[39293] := 16#ED86;
   // UNICODE_TO_GBK[39294] := 16#97F2;
   // UNICODE_TO_GBK[39295] := 16#ED87;
   // UNICODE_TO_GBK[39296] := 16#97F3;
   // UNICODE_TO_GBK[39297] := 16#D2F4;
   // UNICODE_TO_GBK[39298] := 16#97F4;
   // UNICODE_TO_GBK[39299] := 16#ED88;
   // UNICODE_TO_GBK[39300] := 16#97F5;
   // UNICODE_TO_GBK[39301] := 16#D4CF;
   // UNICODE_TO_GBK[39302] := 16#97F6;
   // UNICODE_TO_GBK[39303] := 16#C9D8;
   // UNICODE_TO_GBK[39304] := 16#97F7;
   // UNICODE_TO_GBK[39305] := 16#ED89;
   // UNICODE_TO_GBK[39306] := 16#97F8;
   // UNICODE_TO_GBK[39307] := 16#ED8A;
   // UNICODE_TO_GBK[39308] := 16#97F9;
   // UNICODE_TO_GBK[39309] := 16#ED8B;
   // UNICODE_TO_GBK[39310] := 16#97FA;
   // UNICODE_TO_GBK[39311] := 16#ED8C;
   // UNICODE_TO_GBK[39312] := 16#97FB;
   // UNICODE_TO_GBK[39313] := 16#ED8D;
   // UNICODE_TO_GBK[39314] := 16#97FC;
   // UNICODE_TO_GBK[39315] := 16#ED8E;
   // UNICODE_TO_GBK[39316] := 16#97FD;
   // UNICODE_TO_GBK[39317] := 16#ED8F;
   // UNICODE_TO_GBK[39318] := 16#97FE;
   // UNICODE_TO_GBK[39319] := 16#ED90;
   // UNICODE_TO_GBK[39320] := 16#97FF;
   // UNICODE_TO_GBK[39321] := 16#ED91;
   // UNICODE_TO_GBK[39322] := 16#9800;
   // UNICODE_TO_GBK[39323] := 16#ED92;
   // UNICODE_TO_GBK[39324] := 16#9801;
   // UNICODE_TO_GBK[39325] := 16#ED93;
   // UNICODE_TO_GBK[39326] := 16#9802;
   // UNICODE_TO_GBK[39327] := 16#ED94;
   // UNICODE_TO_GBK[39328] := 16#9803;
   // UNICODE_TO_GBK[39329] := 16#ED95;
   // UNICODE_TO_GBK[39330] := 16#9804;
   // UNICODE_TO_GBK[39331] := 16#ED96;
   // UNICODE_TO_GBK[39332] := 16#9805;
   // UNICODE_TO_GBK[39333] := 16#ED97;
   // UNICODE_TO_GBK[39334] := 16#9806;
   // UNICODE_TO_GBK[39335] := 16#ED98;
   // UNICODE_TO_GBK[39336] := 16#9807;
   // UNICODE_TO_GBK[39337] := 16#ED99;
   // UNICODE_TO_GBK[39338] := 16#9808;
   // UNICODE_TO_GBK[39339] := 16#ED9A;
   // UNICODE_TO_GBK[39340] := 16#9809;
   // UNICODE_TO_GBK[39341] := 16#ED9B;
   // UNICODE_TO_GBK[39342] := 16#980A;
   // UNICODE_TO_GBK[39343] := 16#ED9C;
   // UNICODE_TO_GBK[39344] := 16#980B;
   // UNICODE_TO_GBK[39345] := 16#ED9D;
   // UNICODE_TO_GBK[39346] := 16#980C;
   // UNICODE_TO_GBK[39347] := 16#ED9E;
   // UNICODE_TO_GBK[39348] := 16#980D;
   // UNICODE_TO_GBK[39349] := 16#ED9F;
   // UNICODE_TO_GBK[39350] := 16#980E;
   // UNICODE_TO_GBK[39351] := 16#EDA0;
   // UNICODE_TO_GBK[39352] := 16#980F;
   // UNICODE_TO_GBK[39353] := 16#EE40;
   // UNICODE_TO_GBK[39354] := 16#9810;
   // UNICODE_TO_GBK[39355] := 16#EE41;
   // UNICODE_TO_GBK[39356] := 16#9811;
   // UNICODE_TO_GBK[39357] := 16#EE42;
   // UNICODE_TO_GBK[39358] := 16#9812;
   // UNICODE_TO_GBK[39359] := 16#EE43;
   // UNICODE_TO_GBK[39360] := 16#9813;
   // UNICODE_TO_GBK[39361] := 16#EE44;
   // UNICODE_TO_GBK[39362] := 16#9814;
   // UNICODE_TO_GBK[39363] := 16#EE45;
   // UNICODE_TO_GBK[39364] := 16#9815;
   // UNICODE_TO_GBK[39365] := 16#EE46;
   // UNICODE_TO_GBK[39366] := 16#9816;
   // UNICODE_TO_GBK[39367] := 16#EE47;
   // UNICODE_TO_GBK[39368] := 16#9817;
   // UNICODE_TO_GBK[39369] := 16#EE48;
   // UNICODE_TO_GBK[39370] := 16#9818;
   // UNICODE_TO_GBK[39371] := 16#EE49;
   // UNICODE_TO_GBK[39372] := 16#9819;
   // UNICODE_TO_GBK[39373] := 16#EE4A;
   // UNICODE_TO_GBK[39374] := 16#981A;
   // UNICODE_TO_GBK[39375] := 16#EE4B;
   // UNICODE_TO_GBK[39376] := 16#981B;
   // UNICODE_TO_GBK[39377] := 16#EE4C;
   // UNICODE_TO_GBK[39378] := 16#981C;
   // UNICODE_TO_GBK[39379] := 16#EE4D;
   // UNICODE_TO_GBK[39380] := 16#981D;
   // UNICODE_TO_GBK[39381] := 16#EE4E;
   // UNICODE_TO_GBK[39382] := 16#981E;
   // UNICODE_TO_GBK[39383] := 16#EE4F;
   // UNICODE_TO_GBK[39384] := 16#981F;
   // UNICODE_TO_GBK[39385] := 16#EE50;
   // UNICODE_TO_GBK[39386] := 16#9820;
   // UNICODE_TO_GBK[39387] := 16#EE51;
   // UNICODE_TO_GBK[39388] := 16#9821;
   // UNICODE_TO_GBK[39389] := 16#EE52;
   // UNICODE_TO_GBK[39390] := 16#9822;
   // UNICODE_TO_GBK[39391] := 16#EE53;
   // UNICODE_TO_GBK[39392] := 16#9823;
   // UNICODE_TO_GBK[39393] := 16#EE54;
   // UNICODE_TO_GBK[39394] := 16#9824;
   // UNICODE_TO_GBK[39395] := 16#EE55;
   // UNICODE_TO_GBK[39396] := 16#9825;
   // UNICODE_TO_GBK[39397] := 16#EE56;
   // UNICODE_TO_GBK[39398] := 16#9826;
   // UNICODE_TO_GBK[39399] := 16#EE57;
   // UNICODE_TO_GBK[39400] := 16#9827;
   // UNICODE_TO_GBK[39401] := 16#EE58;
   // UNICODE_TO_GBK[39402] := 16#9828;
   // UNICODE_TO_GBK[39403] := 16#EE59;
   // UNICODE_TO_GBK[39404] := 16#9829;
   // UNICODE_TO_GBK[39405] := 16#EE5A;
   // UNICODE_TO_GBK[39406] := 16#982A;
   // UNICODE_TO_GBK[39407] := 16#EE5B;
   // UNICODE_TO_GBK[39408] := 16#982B;
   // UNICODE_TO_GBK[39409] := 16#EE5C;
   // UNICODE_TO_GBK[39410] := 16#982C;
   // UNICODE_TO_GBK[39411] := 16#EE5D;
   // UNICODE_TO_GBK[39412] := 16#982D;
   // UNICODE_TO_GBK[39413] := 16#EE5E;
   // UNICODE_TO_GBK[39414] := 16#982E;
   // UNICODE_TO_GBK[39415] := 16#EE5F;
   // UNICODE_TO_GBK[39416] := 16#982F;
   // UNICODE_TO_GBK[39417] := 16#EE60;
   // UNICODE_TO_GBK[39418] := 16#9830;
   // UNICODE_TO_GBK[39419] := 16#EE61;
   // UNICODE_TO_GBK[39420] := 16#9831;
   // UNICODE_TO_GBK[39421] := 16#EE62;
   // UNICODE_TO_GBK[39422] := 16#9832;
   // UNICODE_TO_GBK[39423] := 16#EE63;
   // UNICODE_TO_GBK[39424] := 16#9833;
   // UNICODE_TO_GBK[39425] := 16#EE64;
   // UNICODE_TO_GBK[39426] := 16#9834;
   // UNICODE_TO_GBK[39427] := 16#EE65;
   // UNICODE_TO_GBK[39428] := 16#9835;
   // UNICODE_TO_GBK[39429] := 16#EE66;
   // UNICODE_TO_GBK[39430] := 16#9836;
   // UNICODE_TO_GBK[39431] := 16#EE67;
   // UNICODE_TO_GBK[39432] := 16#9837;
   // UNICODE_TO_GBK[39433] := 16#EE68;
   // UNICODE_TO_GBK[39434] := 16#9838;
   // UNICODE_TO_GBK[39435] := 16#EE69;
   // UNICODE_TO_GBK[39436] := 16#9839;
   // UNICODE_TO_GBK[39437] := 16#EE6A;
   // UNICODE_TO_GBK[39438] := 16#983A;
   // UNICODE_TO_GBK[39439] := 16#EE6B;
   // UNICODE_TO_GBK[39440] := 16#983B;
   // UNICODE_TO_GBK[39441] := 16#EE6C;
   // UNICODE_TO_GBK[39442] := 16#983C;
   // UNICODE_TO_GBK[39443] := 16#EE6D;
   // UNICODE_TO_GBK[39444] := 16#983D;
   // UNICODE_TO_GBK[39445] := 16#EE6E;
   // UNICODE_TO_GBK[39446] := 16#983E;
   // UNICODE_TO_GBK[39447] := 16#EE6F;
   // UNICODE_TO_GBK[39448] := 16#983F;
   // UNICODE_TO_GBK[39449] := 16#EE70;
   // UNICODE_TO_GBK[39450] := 16#9840;
   // UNICODE_TO_GBK[39451] := 16#EE71;
   // UNICODE_TO_GBK[39452] := 16#9841;
   // UNICODE_TO_GBK[39453] := 16#EE72;
   // UNICODE_TO_GBK[39454] := 16#9842;
   // UNICODE_TO_GBK[39455] := 16#EE73;
   // UNICODE_TO_GBK[39456] := 16#9843;
   // UNICODE_TO_GBK[39457] := 16#EE74;
   // UNICODE_TO_GBK[39458] := 16#9844;
   // UNICODE_TO_GBK[39459] := 16#EE75;
   // UNICODE_TO_GBK[39460] := 16#9845;
   // UNICODE_TO_GBK[39461] := 16#EE76;
   // UNICODE_TO_GBK[39462] := 16#9846;
   // UNICODE_TO_GBK[39463] := 16#EE77;
   // UNICODE_TO_GBK[39464] := 16#9847;
   // UNICODE_TO_GBK[39465] := 16#EE78;
   // UNICODE_TO_GBK[39466] := 16#9848;
   // UNICODE_TO_GBK[39467] := 16#EE79;
   // UNICODE_TO_GBK[39468] := 16#9849;
   // UNICODE_TO_GBK[39469] := 16#EE7A;
   // UNICODE_TO_GBK[39470] := 16#984A;
   // UNICODE_TO_GBK[39471] := 16#EE7B;
   // UNICODE_TO_GBK[39472] := 16#984B;
   // UNICODE_TO_GBK[39473] := 16#EE7C;
   // UNICODE_TO_GBK[39474] := 16#984C;
   // UNICODE_TO_GBK[39475] := 16#EE7D;
   // UNICODE_TO_GBK[39476] := 16#984D;
   // UNICODE_TO_GBK[39477] := 16#EE7E;
   // UNICODE_TO_GBK[39478] := 16#984E;
   // UNICODE_TO_GBK[39479] := 16#EE80;
   // UNICODE_TO_GBK[39480] := 16#984F;
   // UNICODE_TO_GBK[39481] := 16#EE81;
   // UNICODE_TO_GBK[39482] := 16#9850;
   // UNICODE_TO_GBK[39483] := 16#EE82;
   // UNICODE_TO_GBK[39484] := 16#9851;
   // UNICODE_TO_GBK[39485] := 16#EE83;
   // UNICODE_TO_GBK[39486] := 16#9852;
   // UNICODE_TO_GBK[39487] := 16#EE84;
   // UNICODE_TO_GBK[39488] := 16#9853;
   // UNICODE_TO_GBK[39489] := 16#EE85;
   // UNICODE_TO_GBK[39490] := 16#9854;
   // UNICODE_TO_GBK[39491] := 16#EE86;
   // UNICODE_TO_GBK[39492] := 16#9855;
   // UNICODE_TO_GBK[39493] := 16#EE87;
   // UNICODE_TO_GBK[39494] := 16#9856;
   // UNICODE_TO_GBK[39495] := 16#EE88;
   // UNICODE_TO_GBK[39496] := 16#9857;
   // UNICODE_TO_GBK[39497] := 16#EE89;
   // UNICODE_TO_GBK[39498] := 16#9858;
   // UNICODE_TO_GBK[39499] := 16#EE8A;
   // UNICODE_TO_GBK[39500] := 16#9859;
   // UNICODE_TO_GBK[39501] := 16#EE8B;
   // UNICODE_TO_GBK[39502] := 16#985A;
   // UNICODE_TO_GBK[39503] := 16#EE8C;
   // UNICODE_TO_GBK[39504] := 16#985B;
   // UNICODE_TO_GBK[39505] := 16#EE8D;
   // UNICODE_TO_GBK[39506] := 16#985C;
   // UNICODE_TO_GBK[39507] := 16#EE8E;
   // UNICODE_TO_GBK[39508] := 16#985D;
   // UNICODE_TO_GBK[39509] := 16#EE8F;
   // UNICODE_TO_GBK[39510] := 16#985E;
   // UNICODE_TO_GBK[39511] := 16#EE90;
   // UNICODE_TO_GBK[39512] := 16#985F;
   // UNICODE_TO_GBK[39513] := 16#EE91;
   // UNICODE_TO_GBK[39514] := 16#9860;
   // UNICODE_TO_GBK[39515] := 16#EE92;
   // UNICODE_TO_GBK[39516] := 16#9861;
   // UNICODE_TO_GBK[39517] := 16#EE93;
   // UNICODE_TO_GBK[39518] := 16#9862;
   // UNICODE_TO_GBK[39519] := 16#EE94;
   // UNICODE_TO_GBK[39520] := 16#9863;
   // UNICODE_TO_GBK[39521] := 16#EE95;
   // UNICODE_TO_GBK[39522] := 16#9864;
   // UNICODE_TO_GBK[39523] := 16#EE96;
   // UNICODE_TO_GBK[39524] := 16#9865;
   // UNICODE_TO_GBK[39525] := 16#EE97;
   // UNICODE_TO_GBK[39526] := 16#9866;
   // UNICODE_TO_GBK[39527] := 16#EE98;
   // UNICODE_TO_GBK[39528] := 16#9867;
   // UNICODE_TO_GBK[39529] := 16#EE99;
   // UNICODE_TO_GBK[39530] := 16#9868;
   // UNICODE_TO_GBK[39531] := 16#EE9A;
   // UNICODE_TO_GBK[39532] := 16#9869;
   // UNICODE_TO_GBK[39533] := 16#EE9B;
   // UNICODE_TO_GBK[39534] := 16#986A;
   // UNICODE_TO_GBK[39535] := 16#EE9C;
   // UNICODE_TO_GBK[39536] := 16#986B;
   // UNICODE_TO_GBK[39537] := 16#EE9D;
   // UNICODE_TO_GBK[39538] := 16#986C;
   // UNICODE_TO_GBK[39539] := 16#EE9E;
   // UNICODE_TO_GBK[39540] := 16#986D;
   // UNICODE_TO_GBK[39541] := 16#EE9F;
   // UNICODE_TO_GBK[39542] := 16#986E;
   // UNICODE_TO_GBK[39543] := 16#EEA0;
   // UNICODE_TO_GBK[39544] := 16#986F;
   // UNICODE_TO_GBK[39545] := 16#EF40;
   // UNICODE_TO_GBK[39546] := 16#9870;
   // UNICODE_TO_GBK[39547] := 16#EF41;
   // UNICODE_TO_GBK[39548] := 16#9871;
   // UNICODE_TO_GBK[39549] := 16#EF42;
   // UNICODE_TO_GBK[39550] := 16#9872;
   // UNICODE_TO_GBK[39551] := 16#EF43;
   // UNICODE_TO_GBK[39552] := 16#9873;
   // UNICODE_TO_GBK[39553] := 16#EF44;
   // UNICODE_TO_GBK[39554] := 16#9874;
   // UNICODE_TO_GBK[39555] := 16#EF45;
   // UNICODE_TO_GBK[39556] := 16#9875;
   // UNICODE_TO_GBK[39557] := 16#D2B3;
   // UNICODE_TO_GBK[39558] := 16#9876;
   // UNICODE_TO_GBK[39559] := 16#B6A5;
   // UNICODE_TO_GBK[39560] := 16#9877;
   // UNICODE_TO_GBK[39561] := 16#C7EA;
   // UNICODE_TO_GBK[39562] := 16#9878;
   // UNICODE_TO_GBK[39563] := 16#F1FC;
   // UNICODE_TO_GBK[39564] := 16#9879;
   // UNICODE_TO_GBK[39565] := 16#CFEE;
   // UNICODE_TO_GBK[39566] := 16#987A;
   // UNICODE_TO_GBK[39567] := 16#CBB3;
   // UNICODE_TO_GBK[39568] := 16#987B;
   // UNICODE_TO_GBK[39569] := 16#D0EB;
   // UNICODE_TO_GBK[39570] := 16#987C;
   // UNICODE_TO_GBK[39571] := 16#E7EF;
   // UNICODE_TO_GBK[39572] := 16#987D;
   // UNICODE_TO_GBK[39573] := 16#CDE7;
   // UNICODE_TO_GBK[39574] := 16#987E;
   // UNICODE_TO_GBK[39575] := 16#B9CB;
   // UNICODE_TO_GBK[39576] := 16#987F;
   // UNICODE_TO_GBK[39577] := 16#B6D9;
   // UNICODE_TO_GBK[39578] := 16#9880;
   // UNICODE_TO_GBK[39579] := 16#F1FD;
   // UNICODE_TO_GBK[39580] := 16#9881;
   // UNICODE_TO_GBK[39581] := 16#B0E4;
   // UNICODE_TO_GBK[39582] := 16#9882;
   // UNICODE_TO_GBK[39583] := 16#CBCC;
   // UNICODE_TO_GBK[39584] := 16#9883;
   // UNICODE_TO_GBK[39585] := 16#F1FE;
   // UNICODE_TO_GBK[39586] := 16#9884;
   // UNICODE_TO_GBK[39587] := 16#D4A4;
   // UNICODE_TO_GBK[39588] := 16#9885;
   // UNICODE_TO_GBK[39589] := 16#C2AD;
   // UNICODE_TO_GBK[39590] := 16#9886;
   // UNICODE_TO_GBK[39591] := 16#C1EC;
   // UNICODE_TO_GBK[39592] := 16#9887;
   // UNICODE_TO_GBK[39593] := 16#C6C4;
   // UNICODE_TO_GBK[39594] := 16#9888;
   // UNICODE_TO_GBK[39595] := 16#BEB1;
   // UNICODE_TO_GBK[39596] := 16#9889;
   // UNICODE_TO_GBK[39597] := 16#F2A1;
   // UNICODE_TO_GBK[39598] := 16#988A;
   // UNICODE_TO_GBK[39599] := 16#BCD5;
   // UNICODE_TO_GBK[39600] := 16#988B;
   // UNICODE_TO_GBK[39601] := 16#EF46;
   // UNICODE_TO_GBK[39602] := 16#988C;
   // UNICODE_TO_GBK[39603] := 16#F2A2;
   // UNICODE_TO_GBK[39604] := 16#988D;
   // UNICODE_TO_GBK[39605] := 16#F2A3;
   // UNICODE_TO_GBK[39606] := 16#988E;
   // UNICODE_TO_GBK[39607] := 16#EF47;
   // UNICODE_TO_GBK[39608] := 16#988F;
   // UNICODE_TO_GBK[39609] := 16#F2A4;
   // UNICODE_TO_GBK[39610] := 16#9890;
   // UNICODE_TO_GBK[39611] := 16#D2C3;
   // UNICODE_TO_GBK[39612] := 16#9891;
   // UNICODE_TO_GBK[39613] := 16#C6B5;
   // UNICODE_TO_GBK[39614] := 16#9892;
   // UNICODE_TO_GBK[39615] := 16#EF48;
   // UNICODE_TO_GBK[39616] := 16#9893;
   // UNICODE_TO_GBK[39617] := 16#CDC7;
   // UNICODE_TO_GBK[39618] := 16#9894;
   // UNICODE_TO_GBK[39619] := 16#F2A5;
   // UNICODE_TO_GBK[39620] := 16#9895;
   // UNICODE_TO_GBK[39621] := 16#EF49;
   // UNICODE_TO_GBK[39622] := 16#9896;
   // UNICODE_TO_GBK[39623] := 16#D3B1;
   // UNICODE_TO_GBK[39624] := 16#9897;
   // UNICODE_TO_GBK[39625] := 16#BFC5;
   // UNICODE_TO_GBK[39626] := 16#9898;
   // UNICODE_TO_GBK[39627] := 16#CCE2;
   // UNICODE_TO_GBK[39628] := 16#9899;
   // UNICODE_TO_GBK[39629] := 16#EF4A;
   // UNICODE_TO_GBK[39630] := 16#989A;
   // UNICODE_TO_GBK[39631] := 16#F2A6;
   // UNICODE_TO_GBK[39632] := 16#989B;
   // UNICODE_TO_GBK[39633] := 16#F2A7;
   // UNICODE_TO_GBK[39634] := 16#989C;
   // UNICODE_TO_GBK[39635] := 16#D1D5;
   // UNICODE_TO_GBK[39636] := 16#989D;
   // UNICODE_TO_GBK[39637] := 16#B6EE;
   // UNICODE_TO_GBK[39638] := 16#989E;
   // UNICODE_TO_GBK[39639] := 16#F2A8;
   // UNICODE_TO_GBK[39640] := 16#989F;
   // UNICODE_TO_GBK[39641] := 16#F2A9;
   // UNICODE_TO_GBK[39642] := 16#98A0;
   // UNICODE_TO_GBK[39643] := 16#B5DF;
   // UNICODE_TO_GBK[39644] := 16#98A1;
   // UNICODE_TO_GBK[39645] := 16#F2AA;
   // UNICODE_TO_GBK[39646] := 16#98A2;
   // UNICODE_TO_GBK[39647] := 16#F2AB;
   // UNICODE_TO_GBK[39648] := 16#98A3;
   // UNICODE_TO_GBK[39649] := 16#EF4B;
   // UNICODE_TO_GBK[39650] := 16#98A4;
   // UNICODE_TO_GBK[39651] := 16#B2FC;
   // UNICODE_TO_GBK[39652] := 16#98A5;
   // UNICODE_TO_GBK[39653] := 16#F2AC;
   // UNICODE_TO_GBK[39654] := 16#98A6;
   // UNICODE_TO_GBK[39655] := 16#F2AD;
   // UNICODE_TO_GBK[39656] := 16#98A7;
   // UNICODE_TO_GBK[39657] := 16#C8A7;
   // UNICODE_TO_GBK[39658] := 16#98A8;
   // UNICODE_TO_GBK[39659] := 16#EF4C;
   // UNICODE_TO_GBK[39660] := 16#98A9;
   // UNICODE_TO_GBK[39661] := 16#EF4D;
   // UNICODE_TO_GBK[39662] := 16#98AA;
   // UNICODE_TO_GBK[39663] := 16#EF4E;
   // UNICODE_TO_GBK[39664] := 16#98AB;
   // UNICODE_TO_GBK[39665] := 16#EF4F;
   // UNICODE_TO_GBK[39666] := 16#98AC;
   // UNICODE_TO_GBK[39667] := 16#EF50;
   // UNICODE_TO_GBK[39668] := 16#98AD;
   // UNICODE_TO_GBK[39669] := 16#EF51;
   // UNICODE_TO_GBK[39670] := 16#98AE;
   // UNICODE_TO_GBK[39671] := 16#EF52;
   // UNICODE_TO_GBK[39672] := 16#98AF;
   // UNICODE_TO_GBK[39673] := 16#EF53;
   // UNICODE_TO_GBK[39674] := 16#98B0;
   // UNICODE_TO_GBK[39675] := 16#EF54;
   // UNICODE_TO_GBK[39676] := 16#98B1;
   // UNICODE_TO_GBK[39677] := 16#EF55;
   // UNICODE_TO_GBK[39678] := 16#98B2;
   // UNICODE_TO_GBK[39679] := 16#EF56;
   // UNICODE_TO_GBK[39680] := 16#98B3;
   // UNICODE_TO_GBK[39681] := 16#EF57;
   // UNICODE_TO_GBK[39682] := 16#98B4;
   // UNICODE_TO_GBK[39683] := 16#EF58;
   // UNICODE_TO_GBK[39684] := 16#98B5;
   // UNICODE_TO_GBK[39685] := 16#EF59;
   // UNICODE_TO_GBK[39686] := 16#98B6;
   // UNICODE_TO_GBK[39687] := 16#EF5A;
   // UNICODE_TO_GBK[39688] := 16#98B7;
   // UNICODE_TO_GBK[39689] := 16#EF5B;
   // UNICODE_TO_GBK[39690] := 16#98B8;
   // UNICODE_TO_GBK[39691] := 16#EF5C;
   // UNICODE_TO_GBK[39692] := 16#98B9;
   // UNICODE_TO_GBK[39693] := 16#EF5D;
   // UNICODE_TO_GBK[39694] := 16#98BA;
   // UNICODE_TO_GBK[39695] := 16#EF5E;
   // UNICODE_TO_GBK[39696] := 16#98BB;
   // UNICODE_TO_GBK[39697] := 16#EF5F;
   // UNICODE_TO_GBK[39698] := 16#98BC;
   // UNICODE_TO_GBK[39699] := 16#EF60;
   // UNICODE_TO_GBK[39700] := 16#98BD;
   // UNICODE_TO_GBK[39701] := 16#EF61;
   // UNICODE_TO_GBK[39702] := 16#98BE;
   // UNICODE_TO_GBK[39703] := 16#EF62;
   // UNICODE_TO_GBK[39704] := 16#98BF;
   // UNICODE_TO_GBK[39705] := 16#EF63;
   // UNICODE_TO_GBK[39706] := 16#98C0;
   // UNICODE_TO_GBK[39707] := 16#EF64;
   // UNICODE_TO_GBK[39708] := 16#98C1;
   // UNICODE_TO_GBK[39709] := 16#EF65;
   // UNICODE_TO_GBK[39710] := 16#98C2;
   // UNICODE_TO_GBK[39711] := 16#EF66;
   // UNICODE_TO_GBK[39712] := 16#98C3;
   // UNICODE_TO_GBK[39713] := 16#EF67;
   // UNICODE_TO_GBK[39714] := 16#98C4;
   // UNICODE_TO_GBK[39715] := 16#EF68;
   // UNICODE_TO_GBK[39716] := 16#98C5;
   // UNICODE_TO_GBK[39717] := 16#EF69;
   // UNICODE_TO_GBK[39718] := 16#98C6;
   // UNICODE_TO_GBK[39719] := 16#EF6A;
   // UNICODE_TO_GBK[39720] := 16#98C7;
   // UNICODE_TO_GBK[39721] := 16#EF6B;
   // UNICODE_TO_GBK[39722] := 16#98C8;
   // UNICODE_TO_GBK[39723] := 16#EF6C;
   // UNICODE_TO_GBK[39724] := 16#98C9;
   // UNICODE_TO_GBK[39725] := 16#EF6D;
   // UNICODE_TO_GBK[39726] := 16#98CA;
   // UNICODE_TO_GBK[39727] := 16#EF6E;
   // UNICODE_TO_GBK[39728] := 16#98CB;
   // UNICODE_TO_GBK[39729] := 16#EF6F;
   // UNICODE_TO_GBK[39730] := 16#98CC;
   // UNICODE_TO_GBK[39731] := 16#EF70;
   // UNICODE_TO_GBK[39732] := 16#98CD;
   // UNICODE_TO_GBK[39733] := 16#EF71;
   // UNICODE_TO_GBK[39734] := 16#98CE;
   // UNICODE_TO_GBK[39735] := 16#B7E7;
   // UNICODE_TO_GBK[39736] := 16#98CF;
   // UNICODE_TO_GBK[39737] := 16#EF72;
   // UNICODE_TO_GBK[39738] := 16#98D0;
   // UNICODE_TO_GBK[39739] := 16#EF73;
   // UNICODE_TO_GBK[39740] := 16#98D1;
   // UNICODE_TO_GBK[39741] := 16#ECA9;
   // UNICODE_TO_GBK[39742] := 16#98D2;
   // UNICODE_TO_GBK[39743] := 16#ECAA;
   // UNICODE_TO_GBK[39744] := 16#98D3;
   // UNICODE_TO_GBK[39745] := 16#ECAB;
   // UNICODE_TO_GBK[39746] := 16#98D4;
   // UNICODE_TO_GBK[39747] := 16#EF74;
   // UNICODE_TO_GBK[39748] := 16#98D5;
   // UNICODE_TO_GBK[39749] := 16#ECAC;
   // UNICODE_TO_GBK[39750] := 16#98D6;
   // UNICODE_TO_GBK[39751] := 16#EF75;
   // UNICODE_TO_GBK[39752] := 16#98D7;
   // UNICODE_TO_GBK[39753] := 16#EF76;
   // UNICODE_TO_GBK[39754] := 16#98D8;
   // UNICODE_TO_GBK[39755] := 16#C6AE;
   // UNICODE_TO_GBK[39756] := 16#98D9;
   // UNICODE_TO_GBK[39757] := 16#ECAD;
   // UNICODE_TO_GBK[39758] := 16#98DA;
   // UNICODE_TO_GBK[39759] := 16#ECAE;
   // UNICODE_TO_GBK[39760] := 16#98DB;
   // UNICODE_TO_GBK[39761] := 16#EF77;
   // UNICODE_TO_GBK[39762] := 16#98DC;
   // UNICODE_TO_GBK[39763] := 16#EF78;
   // UNICODE_TO_GBK[39764] := 16#98DD;
   // UNICODE_TO_GBK[39765] := 16#EF79;
   // UNICODE_TO_GBK[39766] := 16#98DE;
   // UNICODE_TO_GBK[39767] := 16#B7C9;
   // UNICODE_TO_GBK[39768] := 16#98DF;
   // UNICODE_TO_GBK[39769] := 16#CAB3;
   // UNICODE_TO_GBK[39770] := 16#98E0;
   // UNICODE_TO_GBK[39771] := 16#EF7A;
   // UNICODE_TO_GBK[39772] := 16#98E1;
   // UNICODE_TO_GBK[39773] := 16#EF7B;
   // UNICODE_TO_GBK[39774] := 16#98E2;
   // UNICODE_TO_GBK[39775] := 16#EF7C;
   // UNICODE_TO_GBK[39776] := 16#98E3;
   // UNICODE_TO_GBK[39777] := 16#EF7D;
   // UNICODE_TO_GBK[39778] := 16#98E4;
   // UNICODE_TO_GBK[39779] := 16#EF7E;
   // UNICODE_TO_GBK[39780] := 16#98E5;
   // UNICODE_TO_GBK[39781] := 16#EF80;
   // UNICODE_TO_GBK[39782] := 16#98E6;
   // UNICODE_TO_GBK[39783] := 16#EF81;
   // UNICODE_TO_GBK[39784] := 16#98E7;
   // UNICODE_TO_GBK[39785] := 16#E2B8;
   // UNICODE_TO_GBK[39786] := 16#98E8;
   // UNICODE_TO_GBK[39787] := 16#F7CF;
   // UNICODE_TO_GBK[39788] := 16#98E9;
   // UNICODE_TO_GBK[39789] := 16#EF82;
   // UNICODE_TO_GBK[39790] := 16#98EA;
   // UNICODE_TO_GBK[39791] := 16#EF83;
   // UNICODE_TO_GBK[39792] := 16#98EB;
   // UNICODE_TO_GBK[39793] := 16#EF84;
   // UNICODE_TO_GBK[39794] := 16#98EC;
   // UNICODE_TO_GBK[39795] := 16#EF85;
   // UNICODE_TO_GBK[39796] := 16#98ED;
   // UNICODE_TO_GBK[39797] := 16#EF86;
   // UNICODE_TO_GBK[39798] := 16#98EE;
   // UNICODE_TO_GBK[39799] := 16#EF87;
   // UNICODE_TO_GBK[39800] := 16#98EF;
   // UNICODE_TO_GBK[39801] := 16#EF88;
   // UNICODE_TO_GBK[39802] := 16#98F0;
   // UNICODE_TO_GBK[39803] := 16#EF89;
   // UNICODE_TO_GBK[39804] := 16#98F1;
   // UNICODE_TO_GBK[39805] := 16#EF8A;
   // UNICODE_TO_GBK[39806] := 16#98F2;
   // UNICODE_TO_GBK[39807] := 16#EF8B;
   // UNICODE_TO_GBK[39808] := 16#98F3;
   // UNICODE_TO_GBK[39809] := 16#EF8C;
   // UNICODE_TO_GBK[39810] := 16#98F4;
   // UNICODE_TO_GBK[39811] := 16#EF8D;
   // UNICODE_TO_GBK[39812] := 16#98F5;
   // UNICODE_TO_GBK[39813] := 16#EF8E;
   // UNICODE_TO_GBK[39814] := 16#98F6;
   // UNICODE_TO_GBK[39815] := 16#EF8F;
   // UNICODE_TO_GBK[39816] := 16#98F7;
   // UNICODE_TO_GBK[39817] := 16#EF90;
   // UNICODE_TO_GBK[39818] := 16#98F8;
   // UNICODE_TO_GBK[39819] := 16#EF91;
   // UNICODE_TO_GBK[39820] := 16#98F9;
   // UNICODE_TO_GBK[39821] := 16#EF92;
   // UNICODE_TO_GBK[39822] := 16#98FA;
   // UNICODE_TO_GBK[39823] := 16#EF93;
   // UNICODE_TO_GBK[39824] := 16#98FB;
   // UNICODE_TO_GBK[39825] := 16#EF94;
